  MoveAbsJ [[135.73,-26.28,-187.24,-106.91,-52.79,56.60],[9E9,9E9,9E9,9E9,9E9,9E9]],speeddata0,DefaultBlend,tool0;
  MoveAbsJ [[136.14,-26.36,-187.04,-105.92,-52.94,56.91],[9E9,9E9,9E9,9E9,9E9,9E9]],speeddata0,DefaultBlend,tool0;
  MoveAbsJ [[136.55,-26.45,-186.84,-104.93,-53.08,57.22],[9E9,9E9,9E9,9E9,9E9,9E9]],speeddata0,DefaultBlend,tool0;
  MoveAbsJ [[136.96,-26.54,-186.65,-103.94,-53.23,57.53],[9E9,9E9,9E9,9E9,9E9,9E9]],speeddata0,DefaultBlend,tool0;
  MoveAbsJ [[137.37,-26.63,-186.45,-102.95,-53.37,57.84],[9E9,9E9,9E9,9E9,9E9,9E9]],speeddata0,DefaultBlend,tool0;
  MoveAbsJ [[137.78,-26.71,-186.25,-101.96,-53.52,58.14],[9E9,9E9,9E9,9E9,9E9,9E9]],speeddata0,DefaultBlend,tool0;
  MoveAbsJ [[138.19,-26.80,-186.05,-100.97,-53.66,58.45],[9E9,9E9,9E9,9E9,9E9,9E9]],speeddata0,DefaultBlend,tool0;
  MoveAbsJ [[138.60,-26.89,-185.85,-99.98,-53.81,58.76],[9E9,9E9,9E9,9E9,9E9,9E9]],speeddata0,DefaultBlend,tool0;
  MoveAbsJ [[139.01,-26.97,-185.66,-98.99,-53.95,59.07],[9E9,9E9,9E9,9E9,9E9,9E9]],speeddata0,DefaultBlend,tool0;
  MoveAbsJ [[139.42,-27.06,-185.46,-98.00,-54.10,59.38],[9E9,9E9,9E9,9E9,9E9,9E9]],speeddata0,DefaultBlend,tool0;
  MoveAbsJ [[139.83,-27.15,-185.26,-97.01,-54.24,59.69],[9E9,9E9,9E9,9E9,9E9,9E9]],speeddata0,DefaultBlend,tool0;
  MoveAbsJ [[140.24,-27.23,-185.06,-96.02,-54.39,60.00],[9E9,9E9,9E9,9E9,9E9,9E9]],speeddata0,DefaultBlend,tool0;
  MoveAbsJ [[140.65,-27.32,-184.86,-95.03,-54.53,60.31],[9E9,9E9,9E9,9E9,9E9,9E9]],speeddata0,DefaultBlend,tool0;
  MoveAbsJ [[141.06,-27.41,-184.67,-94.04,-54.68,60.62],[9E9,9E9,9E9,9E9,9E9,9E9]],speeddata0,DefaultBlend,tool0;
  MoveAbsJ [[141.47,-27.49,-184.47,-93.05,-54.83,60.93],[9E9,9E9,9E9,9E9,9E9,9E9]],speeddata0,DefaultBlend,tool0;
  MoveAbsJ [[141.88,-27.58,-184.27,-92.06,-54.97,61.24],[9E9,9E9,9E9,9E9,9E9,9E9]],speeddata0,DefaultBlend,tool0;
  MoveAbsJ [[142.29,-27.67,-184.07,-91.07,-55.12,61.55],[9E9,9E9,9E9,9E9,9E9,9E9]],speeddata0,DefaultBlend,tool0;
  MoveAbsJ [[142.70,-27.75,-183.87,-90.08,-55.26,61.86],[9E9,9E9,9E9,9E9,9E9,9E9]],speeddata0,DefaultBlend,tool0;
  MoveAbsJ [[143.11,-27.84,-183.68,-89.09,-55.41,62.17],[9E9,9E9,9E9,9E9,9E9,9E9]],speeddata0,DefaultBlend,tool0;
  MoveAbsJ [[143.52,-27.93,-183.48,-88.10,-55.55,62.47],[9E9,9E9,9E9,9E9,9E9,9E9]],speeddata0,DefaultBlend,tool0;
  MoveAbsJ [[143.93,-28.01,-183.28,-87.11,-55.70,62.78],[9E9,9E9,9E9,9E9,9E9,9E9]],speeddata0,DefaultBlend,tool0;
  MoveAbsJ [[144.34,-28.10,-183.08,-86.12,-55.84,63.09],[9E9,9E9,9E9,9E9,9E9,9E9]],speeddata0,DefaultBlend,tool0;
  MoveAbsJ [[144.75,-28.19,-182.88,-85.13,-55.99,63.40],[9E9,9E9,9E9,9E9,9E9,9E9]],speeddata0,DefaultBlend,tool0;
  MoveAbsJ [[145.16,-28.27,-182.69,-84.14,-56.13,63.71],[9E9,9E9,9E9,9E9,9E9,9E9]],speeddata0,DefaultBlend,tool0;
  MoveAbsJ [[145.57,-28.36,-182.49,-83.15,-56.28,64.02],[9E9,9E9,9E9,9E9,9E9,9E9]],speeddata0,DefaultBlend,tool0;
  MoveAbsJ [[145.98,-28.45,-182.29,-82.16,-56.42,64.33],[9E9,9E9,9E9,9E9,9E9,9E9]],speeddata0,DefaultBlend,tool0;
  MoveAbsJ [[146.39,-28.54,-182.09,-81.17,-56.57,64.64],[9E9,9E9,9E9,9E9,9E9,9E9]],speeddata0,DefaultBlend,tool0;
  MoveAbsJ [[146.80,-28.62,-181.90,-80.18,-56.72,64.95],[9E9,9E9,9E9,9E9,9E9,9E9]],speeddata0,DefaultBlend,tool0;
  MoveAbsJ [[147.21,-28.71,-181.70,-79.19,-56.86,65.26],[9E9,9E9,9E9,9E9,9E9,9E9]],speeddata0,DefaultBlend,tool0;
  MoveAbsJ [[147.62,-28.80,-181.50,-78.20,-57.01,65.57],[9E9,9E9,9E9,9E9,9E9,9E9]],speeddata0,DefaultBlend,tool0;
  MoveAbsJ [[148.03,-28.88,-181.30,-77.21,-57.15,65.88],[9E9,9E9,9E9,9E9,9E9,9E9]],speeddata0,DefaultBlend,tool0;
  MoveAbsJ [[148.44,-28.97,-181.10,-76.23,-57.30,66.19],[9E9,9E9,9E9,9E9,9E9,9E9]],speeddata0,DefaultBlend,tool0;
  MoveAbsJ [[148.85,-29.06,-180.91,-75.24,-57.44,66.49],[9E9,9E9,9E9,9E9,9E9,9E9]],speeddata0,DefaultBlend,tool0;
  MoveAbsJ [[149.26,-29.14,-180.71,-74.25,-57.59,66.80],[9E9,9E9,9E9,9E9,9E9,9E9]],speeddata0,DefaultBlend,tool0;
  MoveAbsJ [[149.67,-29.23,-180.51,-73.26,-57.73,67.11],[9E9,9E9,9E9,9E9,9E9,9E9]],speeddata0,DefaultBlend,tool0;
  MoveAbsJ [[150.08,-29.32,-180.31,-72.27,-57.88,67.42],[9E9,9E9,9E9,9E9,9E9,9E9]],speeddata0,DefaultBlend,tool0;
  MoveAbsJ [[150.49,-29.40,-180.11,-71.28,-58.02,67.73],[9E9,9E9,9E9,9E9,9E9,9E9]],speeddata0,DefaultBlend,tool0;
  MoveAbsJ [[150.90,-29.49,-179.92,-70.29,-58.17,68.04],[9E9,9E9,9E9,9E9,9E9,9E9]],speeddata0,DefaultBlend,tool0;
  MoveAbsJ [[151.31,-29.58,-179.72,-69.30,-58.31,68.35],[9E9,9E9,9E9,9E9,9E9,9E9]],speeddata0,DefaultBlend,tool0;
  MoveAbsJ [[151.72,-29.66,-179.52,-68.31,-58.46,68.66],[9E9,9E9,9E9,9E9,9E9,9E9]],speeddata0,DefaultBlend,tool0;
  MoveAbsJ [[152.13,-29.75,-179.32,-67.32,-58.61,68.97],[9E9,9E9,9E9,9E9,9E9,9E9]],speeddata0,DefaultBlend,tool0;
  MoveAbsJ [[152.54,-29.84,-179.12,-66.33,-58.75,69.28],[9E9,9E9,9E9,9E9,9E9,9E9]],speeddata0,DefaultBlend,tool0;
  MoveAbsJ [[152.95,-29.92,-178.93,-65.34,-58.90,69.59],[9E9,9E9,9E9,9E9,9E9,9E9]],speeddata0,DefaultBlend,tool0;
  MoveAbsJ [[153.36,-30.01,-178.73,-64.35,-59.04,69.90],[9E9,9E9,9E9,9E9,9E9,9E9]],speeddata0,DefaultBlend,tool0;
  MoveAbsJ [[153.77,-30.10,-178.53,-63.36,-59.19,70.21],[9E9,9E9,9E9,9E9,9E9,9E9]],speeddata0,DefaultBlend,tool0;
  MoveAbsJ [[154.18,-30.18,-178.33,-62.37,-59.33,70.51],[9E9,9E9,9E9,9E9,9E9,9E9]],speeddata0,DefaultBlend,tool0;
  MoveAbsJ [[154.59,-30.27,-178.13,-61.38,-59.48,70.82],[9E9,9E9,9E9,9E9,9E9,9E9]],speeddata0,DefaultBlend,tool0;
  MoveAbsJ [[155.00,-30.36,-177.94,-60.39,-59.62,71.13],[9E9,9E9,9E9,9E9,9E9,9E9]],speeddata0,DefaultBlend,tool0;
  MoveAbsJ [[155.40,-30.44,-177.74,-59.40,-59.77,71.44],[9E9,9E9,9E9,9E9,9E9,9E9]],speeddata0,DefaultBlend,tool0;
  MoveAbsJ [[155.81,-30.53,-177.54,-58.41,-59.91,71.75],[9E9,9E9,9E9,9E9,9E9,9E9]],speeddata0,DefaultBlend,tool0;
  MoveAbsJ [[156.22,-30.62,-177.34,-57.42,-60.06,72.06],[9E9,9E9,9E9,9E9,9E9,9E9]],speeddata0,DefaultBlend,tool0;
  MoveAbsJ [[156.63,-30.71,-177.14,-56.43,-60.21,72.37],[9E9,9E9,9E9,9E9,9E9,9E9]],speeddata0,DefaultBlend,tool0;
  MoveAbsJ [[157.04,-30.79,-176.95,-55.44,-60.35,72.68],[9E9,9E9,9E9,9E9,9E9,9E9]],speeddata0,DefaultBlend,tool0;
  MoveAbsJ [[157.45,-30.88,-176.75,-54.45,-60.50,72.99],[9E9,9E9,9E9,9E9,9E9,9E9]],speeddata0,DefaultBlend,tool0;
  MoveAbsJ [[157.86,-30.97,-176.55,-53.46,-60.64,73.30],[9E9,9E9,9E9,9E9,9E9,9E9]],speeddata0,DefaultBlend,tool0;
  MoveAbsJ [[158.27,-31.05,-176.35,-52.47,-60.79,73.61],[9E9,9E9,9E9,9E9,9E9,9E9]],speeddata0,DefaultBlend,tool0;
  MoveAbsJ [[158.68,-31.14,-176.16,-51.48,-60.93,73.92],[9E9,9E9,9E9,9E9,9E9,9E9]],speeddata0,DefaultBlend,tool0;
  MoveAbsJ [[159.09,-31.23,-175.96,-50.49,-61.08,74.23],[9E9,9E9,9E9,9E9,9E9,9E9]],speeddata0,DefaultBlend,tool0;
  MoveAbsJ [[159.50,-31.31,-175.76,-49.50,-61.22,74.53],[9E9,9E9,9E9,9E9,9E9,9E9]],speeddata0,DefaultBlend,tool0;
  MoveAbsJ [[159.91,-31.40,-175.56,-48.51,-61.37,74.84],[9E9,9E9,9E9,9E9,9E9,9E9]],speeddata0,DefaultBlend,tool0;
  MoveAbsJ [[160.32,-31.49,-175.36,-47.52,-61.51,75.15],[9E9,9E9,9E9,9E9,9E9,9E9]],speeddata0,DefaultBlend,tool0;
  MoveAbsJ [[160.73,-31.57,-175.17,-46.53,-61.66,75.46],[9E9,9E9,9E9,9E9,9E9,9E9]],speeddata0,DefaultBlend,tool0;
  MoveAbsJ [[161.14,-31.66,-174.97,-45.54,-61.80,75.77],[9E9,9E9,9E9,9E9,9E9,9E9]],speeddata0,DefaultBlend,tool0;
  MoveAbsJ [[161.55,-31.75,-174.77,-44.55,-61.95,76.08],[9E9,9E9,9E9,9E9,9E9,9E9]],speeddata0,DefaultBlend,tool0;
  MoveAbsJ [[161.96,-31.83,-174.57,-43.56,-62.10,76.39],[9E9,9E9,9E9,9E9,9E9,9E9]],speeddata0,DefaultBlend,tool0;
  MoveAbsJ [[162.37,-31.92,-174.37,-42.57,-62.24,76.70],[9E9,9E9,9E9,9E9,9E9,9E9]],speeddata0,DefaultBlend,tool0;
  MoveAbsJ [[162.78,-32.01,-174.18,-41.58,-62.39,77.01],[9E9,9E9,9E9,9E9,9E9,9E9]],speeddata0,DefaultBlend,tool0;
  MoveAbsJ [[163.19,-32.09,-173.98,-40.59,-62.53,77.32],[9E9,9E9,9E9,9E9,9E9,9E9]],speeddata0,DefaultBlend,tool0;
  MoveAbsJ [[163.60,-32.18,-173.78,-39.60,-62.68,77.63],[9E9,9E9,9E9,9E9,9E9,9E9]],speeddata0,DefaultBlend,tool0;
  MoveAbsJ [[164.01,-32.27,-173.58,-38.61,-62.82,77.94],[9E9,9E9,9E9,9E9,9E9,9E9]],speeddata0,DefaultBlend,tool0;
  MoveAbsJ [[164.42,-32.35,-173.38,-37.62,-62.97,78.25],[9E9,9E9,9E9,9E9,9E9,9E9]],speeddata0,DefaultBlend,tool0;
  MoveAbsJ [[164.83,-32.44,-173.19,-36.63,-63.11,78.56],[9E9,9E9,9E9,9E9,9E9,9E9]],speeddata0,DefaultBlend,tool0;
  MoveAbsJ [[165.24,-32.53,-172.99,-35.64,-63.26,78.86],[9E9,9E9,9E9,9E9,9E9,9E9]],speeddata0,DefaultBlend,tool0;
  MoveAbsJ [[165.65,-32.61,-172.79,-34.65,-63.40,79.17],[9E9,9E9,9E9,9E9,9E9,9E9]],speeddata0,DefaultBlend,tool0;
  MoveAbsJ [[166.06,-32.70,-172.59,-33.66,-63.55,79.48],[9E9,9E9,9E9,9E9,9E9,9E9]],speeddata0,DefaultBlend,tool0;
  MoveAbsJ [[166.47,-32.79,-172.39,-32.67,-63.69,79.79],[9E9,9E9,9E9,9E9,9E9,9E9]],speeddata0,DefaultBlend,tool0;
  MoveAbsJ [[166.88,-32.88,-172.20,-31.68,-63.84,80.10],[9E9,9E9,9E9,9E9,9E9,9E9]],speeddata0,DefaultBlend,tool0;
  MoveAbsJ [[167.29,-32.96,-172.00,-30.69,-63.99,80.41],[9E9,9E9,9E9,9E9,9E9,9E9]],speeddata0,DefaultBlend,tool0;
  MoveAbsJ [[167.70,-33.05,-171.80,-29.70,-64.13,80.72],[9E9,9E9,9E9,9E9,9E9,9E9]],speeddata0,DefaultBlend,tool0;
  MoveAbsJ [[168.11,-33.14,-171.60,-28.71,-64.28,81.03],[9E9,9E9,9E9,9E9,9E9,9E9]],speeddata0,DefaultBlend,tool0;
  MoveAbsJ [[168.52,-33.22,-171.40,-27.72,-64.42,81.34],[9E9,9E9,9E9,9E9,9E9,9E9]],speeddata0,DefaultBlend,tool0;
  MoveAbsJ [[168.93,-33.31,-171.21,-26.73,-64.57,81.65],[9E9,9E9,9E9,9E9,9E9,9E9]],speeddata0,DefaultBlend,tool0;
  MoveAbsJ [[169.34,-33.40,-171.01,-25.74,-64.71,81.96],[9E9,9E9,9E9,9E9,9E9,9E9]],speeddata0,DefaultBlend,tool0;
  MoveAbsJ [[169.75,-33.48,-170.81,-24.75,-64.86,82.27],[9E9,9E9,9E9,9E9,9E9,9E9]],speeddata0,DefaultBlend,tool0;
  MoveAbsJ [[170.16,-33.57,-170.61,-23.76,-65.00,82.58],[9E9,9E9,9E9,9E9,9E9,9E9]],speeddata0,DefaultBlend,tool0;
  MoveAbsJ [[170.57,-33.66,-170.42,-22.77,-65.15,82.88],[9E9,9E9,9E9,9E9,9E9,9E9]],speeddata0,DefaultBlend,tool0;
  MoveAbsJ [[170.98,-33.74,-170.22,-21.78,-65.29,83.19],[9E9,9E9,9E9,9E9,9E9,9E9]],speeddata0,DefaultBlend,tool0;
  MoveAbsJ [[171.39,-33.83,-170.02,-20.79,-65.44,83.50],[9E9,9E9,9E9,9E9,9E9,9E9]],speeddata0,DefaultBlend,tool0;
  MoveAbsJ [[171.80,-33.92,-169.82,-19.80,-65.58,83.81],[9E9,9E9,9E9,9E9,9E9,9E9]],speeddata0,DefaultBlend,tool0;
  MoveAbsJ [[172.21,-34.00,-169.62,-18.81,-65.73,84.12],[9E9,9E9,9E9,9E9,9E9,9E9]],speeddata0,DefaultBlend,tool0;
  MoveAbsJ [[172.62,-34.09,-169.43,-17.82,-65.88,84.43],[9E9,9E9,9E9,9E9,9E9,9E9]],speeddata0,DefaultBlend,tool0;
  MoveAbsJ [[173.03,-34.18,-169.23,-16.83,-66.02,84.74],[9E9,9E9,9E9,9E9,9E9,9E9]],speeddata0,DefaultBlend,tool0;
  MoveAbsJ [[173.44,-34.26,-169.03,-15.84,-66.17,85.05],[9E9,9E9,9E9,9E9,9E9,9E9]],speeddata0,DefaultBlend,tool0;
  MoveAbsJ [[173.85,-34.35,-168.83,-14.85,-66.31,85.36],[9E9,9E9,9E9,9E9,9E9,9E9]],speeddata0,DefaultBlend,tool0;
  MoveAbsJ [[174.26,-34.44,-168.63,-13.86,-66.46,85.67],[9E9,9E9,9E9,9E9,9E9,9E9]],speeddata0,DefaultBlend,tool0;
  MoveAbsJ [[174.67,-34.52,-168.44,-12.87,-66.60,85.98],[9E9,9E9,9E9,9E9,9E9,9E9]],speeddata0,DefaultBlend,tool0;
  MoveAbsJ [[175.08,-34.61,-168.24,-11.88,-66.75,86.29],[9E9,9E9,9E9,9E9,9E9,9E9]],speeddata0,DefaultBlend,tool0;
  MoveAbsJ [[175.49,-34.70,-168.04,-10.89,-66.89,86.60],[9E9,9E9,9E9,9E9,9E9,9E9]],speeddata0,DefaultBlend,tool0;
  MoveAbsJ [[175.90,-34.78,-167.84,-9.90,-67.04,86.90],[9E9,9E9,9E9,9E9,9E9,9E9]],speeddata0,DefaultBlend,tool0;
  MoveAbsJ [[176.31,-34.87,-167.64,-8.91,-67.18,87.21],[9E9,9E9,9E9,9E9,9E9,9E9]],speeddata0,DefaultBlend,tool0;
  MoveAbsJ [[176.72,-34.96,-167.45,-7.92,-67.33,87.52],[9E9,9E9,9E9,9E9,9E9,9E9]],speeddata0,DefaultBlend,tool0;
  MoveAbsJ [[177.13,-35.05,-167.25,-6.93,-67.47,87.83],[9E9,9E9,9E9,9E9,9E9,9E9]],speeddata0,DefaultBlend,tool0;
  MoveAbsJ [[177.54,-35.13,-167.05,-5.94,-67.62,88.14],[9E9,9E9,9E9,9E9,9E9,9E9]],speeddata0,DefaultBlend,tool0;
  MoveAbsJ [[177.95,-35.22,-166.85,-4.95,-67.77,88.45],[9E9,9E9,9E9,9E9,9E9,9E9]],speeddata0,DefaultBlend,tool0;
  MoveAbsJ [[178.36,-35.31,-166.65,-3.96,-67.91,88.76],[9E9,9E9,9E9,9E9,9E9,9E9]],speeddata0,DefaultBlend,tool0;
  MoveAbsJ [[178.77,-35.39,-166.46,-2.97,-68.06,89.07],[9E9,9E9,9E9,9E9,9E9,9E9]],speeddata0,DefaultBlend,tool0;
  MoveAbsJ [[179.18,-35.48,-166.26,-1.98,-68.20,89.38],[9E9,9E9,9E9,9E9,9E9,9E9]],speeddata0,DefaultBlend,tool0;
  MoveAbsJ [[179.59,-35.57,-166.06,-0.99,-68.35,89.69],[9E9,9E9,9E9,9E9,9E9,9E9]],speeddata0,DefaultBlend,tool0;
  MoveAbsJ [[180.00,-35.65,-165.86,0.00,-68.49,90.00],[9E9,9E9,9E9,9E9,9E9,9E9]],speeddata0,FinePoint,tool0;
  TPWrite "Action 18 LinearMovement.";
  MoveAbsJ [[180.00,-35.65,-165.86,0.00,-68.49,90.00],[9E9,9E9,9E9,9E9,9E9,9E9]],speeddata0,DefaultBlend,tool0;
  MoveAbsJ [[180.00,-35.59,-165.97,0.00,-68.44,90.00],[9E9,9E9,9E9,9E9,9E9,9E9]],speeddata0,DefaultBlend,tool0;
  MoveAbsJ [[180.00,-36.29,-166.18,0.00,-67.54,90.00],[9E9,9E9,9E9,9E9,9E9,9E9]],speeddata0,DefaultBlend,tool0;
  MoveAbsJ [[180.00,-37.00,-166.36,0.00,-66.64,90.00],[9E9,9E9,9E9,9E9,9E9,9E9]],speeddata0,DefaultBlend,tool0;
  MoveAbsJ [[180.00,-37.73,-166.51,0.00,-65.76,90.00],[9E9,9E9,9E9,9E9,9E9,9E9]],speeddata0,DefaultBlend,tool0;
  MoveAbsJ [[180.00,-38.47,-166.65,0.00,-64.88,90.00],[9E9,9E9,9E9,9E9,9E9,9E9]],speeddata0,DefaultBlend,tool0;
  MoveAbsJ [[180.00,-39.22,-166.76,0.00,-64.02,90.00],[9E9,9E9,9E9,9E9,9E9,9E9]],speeddata0,DefaultBlend,tool0;
  MoveAbsJ [[180.00,-39.99,-166.85,0.00,-63.16,90.00],[9E9,9E9,9E9,9E9,9E9,9E9]],speeddata0,DefaultBlend,tool0;
  MoveAbsJ [[180.00,-40.78,-166.91,0.00,-62.31,90.00],[9E9,9E9,9E9,9E9,9E9,9E9]],speeddata0,DefaultBlend,tool0;
  MoveAbsJ [[180.00,-41.57,-166.96,0.00,-61.47,90.00],[9E9,9E9,9E9,9E9,9E9,9E9]],speeddata0,FinePoint,tool0;
  TPWrite "Action 19 OpenGripper.";
  TPWrite "Press Play to Continue";
  Stop;
  TPWrite "Action 20 LinearMovement.";
  MoveAbsJ [[180.00,-41.57,-166.96,-0.00,-61.47,90.00],[9E9,9E9,9E9,9E9,9E9,9E9]],speeddata0,DefaultBlend,tool0;
  MoveAbsJ [[180.00,-40.78,-166.92,0.00,-62.30,90.00],[9E9,9E9,9E9,9E9,9E9,9E9]],speeddata0,DefaultBlend,tool0;
  MoveAbsJ [[180.00,-39.99,-166.86,0.00,-63.14,90.00],[9E9,9E9,9E9,9E9,9E9,9E9]],speeddata0,DefaultBlend,tool0;
  MoveAbsJ [[180.00,-39.22,-166.78,0.00,-64.00,90.00],[9E9,9E9,9E9,9E9,9E9,9E9]],speeddata0,DefaultBlend,tool0;
  MoveAbsJ [[180.00,-38.46,-166.67,0.00,-64.86,90.00],[9E9,9E9,9E9,9E9,9E9,9E9]],speeddata0,DefaultBlend,tool0;
  MoveAbsJ [[180.00,-37.72,-166.54,0.00,-65.74,90.00],[9E9,9E9,9E9,9E9,9E9,9E9]],speeddata0,DefaultBlend,tool0;
  MoveAbsJ [[180.00,-36.99,-166.39,0.00,-66.63,90.00],[9E9,9E9,9E9,9E9,9E9,9E9]],speeddata0,DefaultBlend,tool0;
  MoveAbsJ [[180.00,-36.27,-166.21,0.00,-67.52,90.00],[9E9,9E9,9E9,9E9,9E9,9E9]],speeddata0,DefaultBlend,tool0;
  MoveAbsJ [[180.00,-35.58,-166.00,0.00,-68.42,90.00],[9E9,9E9,9E9,9E9,9E9,9E9]],speeddata0,FinePoint,tool0;
  TPWrite "Action 21 FreeMovement.";
  MoveAbsJ [[180.00,-35.58,-166.00,0.00,-68.42,90.00],[9E9,9E9,9E9,9E9,9E9,9E9]],speeddata0,DefaultBlend,tool0;
  MoveAbsJ [[179.59,-35.49,-166.20,-0.99,-68.28,89.69],[9E9,9E9,9E9,9E9,9E9,9E9]],speeddata0,DefaultBlend,tool0;
  MoveAbsJ [[179.18,-35.40,-166.40,-1.98,-68.13,89.38],[9E9,9E9,9E9,9E9,9E9,9E9]],speeddata0,DefaultBlend,tool0;
  MoveAbsJ [[178.77,-35.32,-166.59,-2.97,-67.99,89.07],[9E9,9E9,9E9,9E9,9E9,9E9]],speeddata0,DefaultBlend,tool0;
  MoveAbsJ [[178.36,-35.23,-166.79,-3.96,-67.84,88.76],[9E9,9E9,9E9,9E9,9E9,9E9]],speeddata0,DefaultBlend,tool0;
  MoveAbsJ [[177.95,-35.14,-166.99,-4.95,-67.70,88.45],[9E9,9E9,9E9,9E9,9E9,9E9]],speeddata0,DefaultBlend,tool0;
  MoveAbsJ [[177.54,-35.06,-167.18,-5.94,-67.55,88.14],[9E9,9E9,9E9,9E9,9E9,9E9]],speeddata0,DefaultBlend,tool0;
  MoveAbsJ [[177.13,-34.97,-167.38,-6.93,-67.41,87.83],[9E9,9E9,9E9,9E9,9E9,9E9]],speeddata0,DefaultBlend,tool0;
  MoveAbsJ [[176.72,-34.89,-167.58,-7.92,-67.26,87.52],[9E9,9E9,9E9,9E9,9E9,9E9]],speeddata0,DefaultBlend,tool0;
  MoveAbsJ [[176.31,-34.80,-167.77,-8.91,-67.12,87.21],[9E9,9E9,9E9,9E9,9E9,9E9]],speeddata0,DefaultBlend,tool0;
  MoveAbsJ [[175.90,-34.71,-167.97,-9.90,-66.97,86.91],[9E9,9E9,9E9,9E9,9E9,9E9]],speeddata0,DefaultBlend,tool0;
  MoveAbsJ [[175.49,-34.63,-168.17,-10.89,-66.83,86.60],[9E9,9E9,9E9,9E9,9E9,9E9]],speeddata0,DefaultBlend,tool0;
  MoveAbsJ [[175.08,-34.54,-168.36,-11.88,-66.68,86.29],[9E9,9E9,9E9,9E9,9E9,9E9]],speeddata0,DefaultBlend,tool0;
  MoveAbsJ [[174.67,-34.45,-168.56,-12.87,-66.54,85.98],[9E9,9E9,9E9,9E9,9E9,9E9]],speeddata0,DefaultBlend,tool0;
  MoveAbsJ [[174.26,-34.37,-168.76,-13.86,-66.39,85.67],[9E9,9E9,9E9,9E9,9E9,9E9]],speeddata0,DefaultBlend,tool0;
  MoveAbsJ [[173.85,-34.28,-168.95,-14.85,-66.25,85.36],[9E9,9E9,9E9,9E9,9E9,9E9]],speeddata0,DefaultBlend,tool0;
  MoveAbsJ [[173.44,-34.20,-169.15,-15.84,-66.10,85.05],[9E9,9E9,9E9,9E9,9E9,9E9]],speeddata0,DefaultBlend,tool0;
  MoveAbsJ [[173.03,-34.11,-169.35,-16.83,-65.96,84.74],[9E9,9E9,9E9,9E9,9E9,9E9]],speeddata0,DefaultBlend,tool0;
  MoveAbsJ [[172.62,-34.02,-169.54,-17.82,-65.81,84.43],[9E9,9E9,9E9,9E9,9E9,9E9]],speeddata0,DefaultBlend,tool0;
  MoveAbsJ [[172.21,-33.94,-169.74,-18.81,-65.67,84.12],[9E9,9E9,9E9,9E9,9E9,9E9]],speeddata0,DefaultBlend,tool0;
  MoveAbsJ [[171.80,-33.85,-169.94,-19.80,-65.52,83.81],[9E9,9E9,9E9,9E9,9E9,9E9]],speeddata0,DefaultBlend,tool0;
  MoveAbsJ [[171.39,-33.76,-170.13,-20.78,-65.38,83.50],[9E9,9E9,9E9,9E9,9E9,9E9]],speeddata0,DefaultBlend,tool0;
  MoveAbsJ [[170.98,-33.68,-170.33,-21.77,-65.23,83.19],[9E9,9E9,9E9,9E9,9E9,9E9]],speeddata0,DefaultBlend,tool0;
  MoveAbsJ [[170.57,-33.59,-170.53,-22.76,-65.09,82.88],[9E9,9E9,9E9,9E9,9E9,9E9]],speeddata0,DefaultBlend,tool0;
  MoveAbsJ [[170.16,-33.51,-170.73,-23.75,-64.94,82.57],[9E9,9E9,9E9,9E9,9E9,9E9]],speeddata0,DefaultBlend,tool0;
  MoveAbsJ [[169.75,-33.42,-170.92,-24.74,-64.80,82.26],[9E9,9E9,9E9,9E9,9E9,9E9]],speeddata0,DefaultBlend,tool0;
  MoveAbsJ [[169.34,-33.33,-171.12,-25.73,-64.65,81.95],[9E9,9E9,9E9,9E9,9E9,9E9]],speeddata0,DefaultBlend,tool0;
  MoveAbsJ [[168.93,-33.25,-171.32,-26.72,-64.51,81.64],[9E9,9E9,9E9,9E9,9E9,9E9]],speeddata0,DefaultBlend,tool0;
  MoveAbsJ [[168.53,-33.16,-171.51,-27.71,-64.36,81.34],[9E9,9E9,9E9,9E9,9E9,9E9]],speeddata0,DefaultBlend,tool0;
  MoveAbsJ [[168.12,-33.07,-171.71,-28.70,-64.22,81.03],[9E9,9E9,9E9,9E9,9E9,9E9]],speeddata0,DefaultBlend,tool0;
  MoveAbsJ [[167.71,-32.99,-171.91,-29.69,-64.08,80.72],[9E9,9E9,9E9,9E9,9E9,9E9]],speeddata0,DefaultBlend,tool0;
  MoveAbsJ [[167.30,-32.90,-172.10,-30.68,-63.93,80.41],[9E9,9E9,9E9,9E9,9E9,9E9]],speeddata0,DefaultBlend,tool0;
  MoveAbsJ [[166.89,-32.82,-172.30,-31.67,-63.79,80.10],[9E9,9E9,9E9,9E9,9E9,9E9]],speeddata0,DefaultBlend,tool0;
  MoveAbsJ [[166.48,-32.73,-172.50,-32.66,-63.64,79.79],[9E9,9E9,9E9,9E9,9E9,9E9]],speeddata0,DefaultBlend,tool0;
  MoveAbsJ [[166.07,-32.64,-172.69,-33.65,-63.50,79.48],[9E9,9E9,9E9,9E9,9E9,9E9]],speeddata0,DefaultBlend,tool0;
  MoveAbsJ [[165.66,-32.56,-172.89,-34.64,-63.35,79.17],[9E9,9E9,9E9,9E9,9E9,9E9]],speeddata0,DefaultBlend,tool0;
  MoveAbsJ [[165.25,-32.47,-173.09,-35.63,-63.21,78.86],[9E9,9E9,9E9,9E9,9E9,9E9]],speeddata0,DefaultBlend,tool0;
  MoveAbsJ [[164.84,-32.38,-173.28,-36.62,-63.06,78.55],[9E9,9E9,9E9,9E9,9E9,9E9]],speeddata0,DefaultBlend,tool0;
  MoveAbsJ [[164.43,-32.30,-173.48,-37.61,-62.92,78.24],[9E9,9E9,9E9,9E9,9E9,9E9]],speeddata0,DefaultBlend,tool0;
  MoveAbsJ [[164.02,-32.21,-173.68,-38.60,-62.77,77.93],[9E9,9E9,9E9,9E9,9E9,9E9]],speeddata0,DefaultBlend,tool0;
  MoveAbsJ [[163.61,-32.13,-173.87,-39.59,-62.63,77.62],[9E9,9E9,9E9,9E9,9E9,9E9]],speeddata0,DefaultBlend,tool0;
  MoveAbsJ [[163.20,-32.04,-174.07,-40.58,-62.48,77.31],[9E9,9E9,9E9,9E9,9E9,9E9]],speeddata0,DefaultBlend,tool0;
  MoveAbsJ [[162.79,-31.95,-174.27,-41.57,-62.34,77.00],[9E9,9E9,9E9,9E9,9E9,9E9]],speeddata0,DefaultBlend,tool0;
  MoveAbsJ [[162.38,-31.87,-174.46,-42.56,-62.19,76.69],[9E9,9E9,9E9,9E9,9E9,9E9]],speeddata0,DefaultBlend,tool0;
  MoveAbsJ [[161.97,-31.78,-174.66,-43.55,-62.05,76.38],[9E9,9E9,9E9,9E9,9E9,9E9]],speeddata0,DefaultBlend,tool0;
  MoveAbsJ [[161.56,-31.69,-174.86,-44.54,-61.90,76.07],[9E9,9E9,9E9,9E9,9E9,9E9]],speeddata0,DefaultBlend,tool0;
  MoveAbsJ [[161.15,-31.61,-175.05,-45.53,-61.76,75.76],[9E9,9E9,9E9,9E9,9E9,9E9]],speeddata0,DefaultBlend,tool0;
  MoveAbsJ [[160.74,-31.52,-175.25,-46.52,-61.61,75.46],[9E9,9E9,9E9,9E9,9E9,9E9]],speeddata0,DefaultBlend,tool0;
  MoveAbsJ [[160.33,-31.44,-175.45,-47.51,-61.47,75.15],[9E9,9E9,9E9,9E9,9E9,9E9]],speeddata0,DefaultBlend,tool0;
  MoveAbsJ [[159.92,-31.35,-175.64,-48.50,-61.32,74.84],[9E9,9E9,9E9,9E9,9E9,9E9]],speeddata0,DefaultBlend,tool0;
  MoveAbsJ [[159.51,-31.26,-175.84,-49.49,-61.18,74.53],[9E9,9E9,9E9,9E9,9E9,9E9]],speeddata0,DefaultBlend,tool0;
  MoveAbsJ [[159.10,-31.18,-176.04,-50.48,-61.03,74.22],[9E9,9E9,9E9,9E9,9E9,9E9]],speeddata0,DefaultBlend,tool0;
  MoveAbsJ [[158.69,-31.09,-176.24,-51.47,-60.89,73.91],[9E9,9E9,9E9,9E9,9E9,9E9]],speeddata0,DefaultBlend,tool0;
  MoveAbsJ [[158.28,-31.00,-176.43,-52.46,-60.74,73.60],[9E9,9E9,9E9,9E9,9E9,9E9]],speeddata0,DefaultBlend,tool0;
  MoveAbsJ [[157.87,-30.92,-176.63,-53.45,-60.60,73.29],[9E9,9E9,9E9,9E9,9E9,9E9]],speeddata0,DefaultBlend,tool0;
  MoveAbsJ [[157.46,-30.83,-176.83,-54.44,-60.45,72.98],[9E9,9E9,9E9,9E9,9E9,9E9]],speeddata0,DefaultBlend,tool0;
  MoveAbsJ [[157.05,-30.75,-177.02,-55.43,-60.31,72.67],[9E9,9E9,9E9,9E9,9E9,9E9]],speeddata0,DefaultBlend,tool0;
  MoveAbsJ [[156.64,-30.66,-177.22,-56.42,-60.16,72.36],[9E9,9E9,9E9,9E9,9E9,9E9]],speeddata0,DefaultBlend,tool0;
  MoveAbsJ [[156.23,-30.57,-177.42,-57.41,-60.02,72.05],[9E9,9E9,9E9,9E9,9E9,9E9]],speeddata0,DefaultBlend,tool0;
  MoveAbsJ [[155.82,-30.49,-177.61,-58.40,-59.87,71.74],[9E9,9E9,9E9,9E9,9E9,9E9]],speeddata0,DefaultBlend,tool0;
  MoveAbsJ [[155.41,-30.40,-177.81,-59.39,-59.73,71.43],[9E9,9E9,9E9,9E9,9E9,9E9]],speeddata0,DefaultBlend,tool0;
  MoveAbsJ [[155.00,-30.31,-178.01,-60.38,-59.58,71.12],[9E9,9E9,9E9,9E9,9E9,9E9]],speeddata0,DefaultBlend,tool0;
  MoveAbsJ [[154.59,-30.23,-178.20,-61.36,-59.44,70.81],[9E9,9E9,9E9,9E9,9E9,9E9]],speeddata0,DefaultBlend,tool0;
  MoveAbsJ [[154.18,-30.14,-178.40,-62.35,-59.29,70.50],[9E9,9E9,9E9,9E9,9E9,9E9]],speeddata0,DefaultBlend,tool0;
  MoveAbsJ [[153.77,-30.06,-178.60,-63.34,-59.15,70.19],[9E9,9E9,9E9,9E9,9E9,9E9]],speeddata0,DefaultBlend,tool0;
  MoveAbsJ [[153.36,-29.97,-178.79,-64.33,-59.01,69.89],[9E9,9E9,9E9,9E9,9E9,9E9]],speeddata0,DefaultBlend,tool0;
  MoveAbsJ [[152.95,-29.88,-178.99,-65.32,-58.86,69.58],[9E9,9E9,9E9,9E9,9E9,9E9]],speeddata0,DefaultBlend,tool0;
  MoveAbsJ [[152.54,-29.80,-179.19,-66.31,-58.72,69.27],[9E9,9E9,9E9,9E9,9E9,9E9]],speeddata0,DefaultBlend,tool0;
  MoveAbsJ [[152.13,-29.71,-179.38,-67.30,-58.57,68.96],[9E9,9E9,9E9,9E9,9E9,9E9]],speeddata0,DefaultBlend,tool0;
  MoveAbsJ [[151.72,-29.62,-179.58,-68.29,-58.43,68.65],[9E9,9E9,9E9,9E9,9E9,9E9]],speeddata0,DefaultBlend,tool0;
  MoveAbsJ [[151.31,-29.54,-179.78,-69.28,-58.28,68.34],[9E9,9E9,9E9,9E9,9E9,9E9]],speeddata0,DefaultBlend,tool0;
  MoveAbsJ [[150.90,-29.45,-179.97,-70.27,-58.14,68.03],[9E9,9E9,9E9,9E9,9E9,9E9]],speeddata0,DefaultBlend,tool0;
  MoveAbsJ [[150.49,-29.37,-180.17,-71.26,-57.99,67.72],[9E9,9E9,9E9,9E9,9E9,9E9]],speeddata0,DefaultBlend,tool0;
  MoveAbsJ [[150.08,-29.28,-180.37,-72.25,-57.85,67.41],[9E9,9E9,9E9,9E9,9E9,9E9]],speeddata0,DefaultBlend,tool0;
  MoveAbsJ [[149.67,-29.19,-180.56,-73.24,-57.70,67.10],[9E9,9E9,9E9,9E9,9E9,9E9]],speeddata0,DefaultBlend,tool0;
  MoveAbsJ [[149.26,-29.11,-180.76,-74.23,-57.56,66.79],[9E9,9E9,9E9,9E9,9E9,9E9]],speeddata0,DefaultBlend,tool0;
  MoveAbsJ [[148.85,-29.02,-180.96,-75.22,-57.41,66.48],[9E9,9E9,9E9,9E9,9E9,9E9]],speeddata0,DefaultBlend,tool0;
  MoveAbsJ [[148.44,-28.93,-181.15,-76.21,-57.27,66.17],[9E9,9E9,9E9,9E9,9E9,9E9]],speeddata0,DefaultBlend,tool0;
  MoveAbsJ [[148.03,-28.85,-181.35,-77.20,-57.12,65.86],[9E9,9E9,9E9,9E9,9E9,9E9]],speeddata0,DefaultBlend,tool0;
  MoveAbsJ [[147.62,-28.76,-181.55,-78.19,-56.98,65.55],[9E9,9E9,9E9,9E9,9E9,9E9]],speeddata0,DefaultBlend,tool0;
  MoveAbsJ [[147.21,-28.68,-181.75,-79.18,-56.83,65.24],[9E9,9E9,9E9,9E9,9E9,9E9]],speeddata0,DefaultBlend,tool0;
  MoveAbsJ [[146.80,-28.59,-181.94,-80.17,-56.69,64.93],[9E9,9E9,9E9,9E9,9E9,9E9]],speeddata0,DefaultBlend,tool0;
  MoveAbsJ [[146.39,-28.50,-182.14,-81.16,-56.54,64.62],[9E9,9E9,9E9,9E9,9E9,9E9]],speeddata0,DefaultBlend,tool0;
  MoveAbsJ [[145.98,-28.42,-182.34,-82.15,-56.40,64.31],[9E9,9E9,9E9,9E9,9E9,9E9]],speeddata0,DefaultBlend,tool0;
  MoveAbsJ [[145.58,-28.33,-182.53,-83.14,-56.25,64.01],[9E9,9E9,9E9,9E9,9E9,9E9]],speeddata0,DefaultBlend,tool0;
  MoveAbsJ [[145.17,-28.24,-182.73,-84.13,-56.11,63.70],[9E9,9E9,9E9,9E9,9E9,9E9]],speeddata0,DefaultBlend,tool0;
  MoveAbsJ [[144.76,-28.16,-182.93,-85.12,-55.96,63.39],[9E9,9E9,9E9,9E9,9E9,9E9]],speeddata0,DefaultBlend,tool0;
  MoveAbsJ [[144.35,-28.07,-183.12,-86.11,-55.82,63.08],[9E9,9E9,9E9,9E9,9E9,9E9]],speeddata0,DefaultBlend,tool0;
  MoveAbsJ [[143.94,-27.99,-183.32,-87.10,-55.67,62.77],[9E9,9E9,9E9,9E9,9E9,9E9]],speeddata0,DefaultBlend,tool0;
  MoveAbsJ [[143.53,-27.90,-183.52,-88.09,-55.53,62.46],[9E9,9E9,9E9,9E9,9E9,9E9]],speeddata0,DefaultBlend,tool0;
  MoveAbsJ [[143.12,-27.81,-183.71,-89.08,-55.38,62.15],[9E9,9E9,9E9,9E9,9E9,9E9]],speeddata0,DefaultBlend,tool0;
  MoveAbsJ [[142.71,-27.73,-183.91,-90.07,-55.24,61.84],[9E9,9E9,9E9,9E9,9E9,9E9]],speeddata0,DefaultBlend,tool0;
  MoveAbsJ [[142.30,-27.64,-184.11,-91.06,-55.09,61.53],[9E9,9E9,9E9,9E9,9E9,9E9]],speeddata0,DefaultBlend,tool0;
  MoveAbsJ [[141.89,-27.55,-184.30,-92.05,-54.95,61.22],[9E9,9E9,9E9,9E9,9E9,9E9]],speeddata0,DefaultBlend,tool0;
  MoveAbsJ [[141.48,-27.47,-184.50,-93.04,-54.80,60.91],[9E9,9E9,9E9,9E9,9E9,9E9]],speeddata0,DefaultBlend,tool0;
  MoveAbsJ [[141.07,-27.38,-184.70,-94.03,-54.66,60.60],[9E9,9E9,9E9,9E9,9E9,9E9]],speeddata0,DefaultBlend,tool0;
  MoveAbsJ [[140.66,-27.30,-184.89,-95.02,-54.51,60.29],[9E9,9E9,9E9,9E9,9E9,9E9]],speeddata0,DefaultBlend,tool0;
  MoveAbsJ [[140.25,-27.21,-185.09,-96.01,-54.37,59.98],[9E9,9E9,9E9,9E9,9E9,9E9]],speeddata0,DefaultBlend,tool0;
  MoveAbsJ [[139.84,-27.12,-185.29,-97.00,-54.22,59.67],[9E9,9E9,9E9,9E9,9E9,9E9]],speeddata0,DefaultBlend,tool0;
  MoveAbsJ [[139.43,-27.04,-185.48,-97.99,-54.08,59.36],[9E9,9E9,9E9,9E9,9E9,9E9]],speeddata0,DefaultBlend,tool0;
  MoveAbsJ [[139.02,-26.95,-185.68,-98.98,-53.94,59.05],[9E9,9E9,9E9,9E9,9E9,9E9]],speeddata0,DefaultBlend,tool0;
  MoveAbsJ [[138.61,-26.86,-185.88,-99.97,-53.79,58.74],[9E9,9E9,9E9,9E9,9E9,9E9]],speeddata0,DefaultBlend,tool0;
  MoveAbsJ [[138.20,-26.78,-186.07,-100.96,-53.65,58.44],[9E9,9E9,9E9,9E9,9E9,9E9]],speeddata0,DefaultBlend,tool0;
  MoveAbsJ [[137.79,-26.69,-186.27,-101.95,-53.50,58.13],[9E9,9E9,9E9,9E9,9E9,9E9]],speeddata0,DefaultBlend,tool0;
  MoveAbsJ [[137.38,-26.61,-186.47,-102.93,-53.36,57.82],[9E9,9E9,9E9,9E9,9E9,9E9]],speeddata0,DefaultBlend,tool0;
  MoveAbsJ [[136.97,-26.52,-186.66,-103.92,-53.21,57.51],[9E9,9E9,9E9,9E9,9E9,9E9]],speeddata0,DefaultBlend,tool0;
  MoveAbsJ [[136.56,-26.43,-186.86,-104.91,-53.07,57.20],[9E9,9E9,9E9,9E9,9E9,9E9]],speeddata0,DefaultBlend,tool0;
  MoveAbsJ [[136.15,-26.35,-187.06,-105.90,-52.92,56.89],[9E9,9E9,9E9,9E9,9E9,9E9]],speeddata0,DefaultBlend,tool0;
  MoveAbsJ [[135.74,-26.26,-187.26,-106.89,-52.78,56.58],[9E9,9E9,9E9,9E9,9E9,9E9]],speeddata0,DefaultBlend,tool0;
  MoveAbsJ [[135.33,-26.17,-187.45,-107.88,-52.63,56.27],[9E9,9E9,9E9,9E9,9E9,9E9]],speeddata0,DefaultBlend,tool0;
  MoveAbsJ [[134.92,-26.09,-187.65,-108.87,-52.49,55.96],[9E9,9E9,9E9,9E9,9E9,9E9]],speeddata0,DefaultBlend,tool0;
  MoveAbsJ [[134.51,-26.00,-187.85,-109.86,-52.34,55.65],[9E9,9E9,9E9,9E9,9E9,9E9]],speeddata0,DefaultBlend,tool0;
  MoveAbsJ [[134.10,-25.92,-188.04,-110.85,-52.20,55.34],[9E9,9E9,9E9,9E9,9E9,9E9]],speeddata0,DefaultBlend,tool0;
  MoveAbsJ [[133.69,-25.83,-188.24,-111.84,-52.05,55.03],[9E9,9E9,9E9,9E9,9E9,9E9]],speeddata0,DefaultBlend,tool0;
  MoveAbsJ [[133.28,-25.74,-188.44,-112.83,-51.91,54.72],[9E9,9E9,9E9,9E9,9E9,9E9]],speeddata0,DefaultBlend,tool0;
  MoveAbsJ [[132.87,-25.66,-188.63,-113.82,-51.76,54.41],[9E9,9E9,9E9,9E9,9E9,9E9]],speeddata0,DefaultBlend,tool0;
  MoveAbsJ [[132.46,-25.57,-188.83,-114.81,-51.62,54.10],[9E9,9E9,9E9,9E9,9E9,9E9]],speeddata0,DefaultBlend,tool0;
  MoveAbsJ [[132.05,-25.48,-189.03,-115.80,-51.47,53.79],[9E9,9E9,9E9,9E9,9E9,9E9]],speeddata0,DefaultBlend,tool0;
  MoveAbsJ [[131.64,-25.40,-189.22,-116.79,-51.33,53.48],[9E9,9E9,9E9,9E9,9E9,9E9]],speeddata0,DefaultBlend,tool0;
  MoveAbsJ [[131.23,-25.31,-189.42,-117.78,-51.18,53.17],[9E9,9E9,9E9,9E9,9E9,9E9]],speeddata0,DefaultBlend,tool0;
  MoveAbsJ [[130.82,-25.23,-189.62,-118.77,-51.04,52.87],[9E9,9E9,9E9,9E9,9E9,9E9]],speeddata0,DefaultBlend,tool0;
  MoveAbsJ [[130.41,-25.14,-189.81,-119.76,-50.89,52.56],[9E9,9E9,9E9,9E9,9E9,9E9]],speeddata0,DefaultBlend,tool0;
  MoveAbsJ [[130.00,-25.05,-190.01,-120.75,-50.75,52.25],[9E9,9E9,9E9,9E9,9E9,9E9]],speeddata0,DefaultBlend,tool0;
  MoveAbsJ [[129.59,-24.97,-190.21,-121.74,-50.60,51.94],[9E9,9E9,9E9,9E9,9E9,9E9]],speeddata0,DefaultBlend,tool0;
  MoveAbsJ [[129.18,-24.88,-190.40,-122.73,-50.46,51.63],[9E9,9E9,9E9,9E9,9E9,9E9]],speeddata0,DefaultBlend,tool0;
  MoveAbsJ [[128.77,-24.79,-190.60,-123.72,-50.31,51.32],[9E9,9E9,9E9,9E9,9E9,9E9]],speeddata0,DefaultBlend,tool0;
  MoveAbsJ [[128.36,-24.71,-190.80,-124.71,-50.17,51.01],[9E9,9E9,9E9,9E9,9E9,9E9]],speeddata0,DefaultBlend,tool0;
  MoveAbsJ [[127.95,-24.62,-190.99,-125.70,-50.02,50.70],[9E9,9E9,9E9,9E9,9E9,9E9]],speeddata0,DefaultBlend,tool0;
  MoveAbsJ [[127.54,-24.54,-191.19,-126.69,-49.88,50.39],[9E9,9E9,9E9,9E9,9E9,9E9]],speeddata0,DefaultBlend,tool0;
  MoveAbsJ [[127.13,-24.45,-191.39,-127.68,-49.73,50.08],[9E9,9E9,9E9,9E9,9E9,9E9]],speeddata0,FinePoint,tool0;
  TPWrite "Action 22 LoadWorkpiece.";
  TPWrite "Press Play to Continue";
  Stop;
  TPWrite "Action 23 CloseGripper.";
  TPWrite "Press Play to Continue";
  Stop;
  TPWrite "Action 24 FreeMovement.";
  MoveAbsJ [[127.13,-24.45,-191.39,-127.68,-49.73,50.08],[9E9,9E9,9E9,9E9,9E9,9E9]],speeddata0,DefaultBlend,tool0;
  MoveAbsJ [[126.87,-24.11,-191.00,-127.69,-49.49,49.58],[9E9,9E9,9E9,9E9,9E9,9E9]],speeddata0,DefaultBlend,tool0;
  MoveAbsJ [[126.65,-23.69,-190.02,-127.13,-49.25,48.92],[9E9,9E9,9E9,9E9,9E9,9E9]],speeddata0,DefaultBlend,tool0;
  MoveAbsJ [[126.94,-23.83,-189.31,-126.15,-49.43,49.02],[9E9,9E9,9E9,9E9,9E9,9E9]],speeddata0,DefaultBlend,tool0;
  MoveAbsJ [[127.23,-23.96,-188.61,-125.17,-49.62,49.11],[9E9,9E9,9E9,9E9,9E9,9E9]],speeddata0,DefaultBlend,tool0;
  MoveAbsJ [[127.53,-24.10,-187.90,-124.19,-49.81,49.21],[9E9,9E9,9E9,9E9,9E9,9E9]],speeddata0,DefaultBlend,tool0;
  MoveAbsJ [[127.82,-24.24,-187.19,-123.21,-50.00,49.30],[9E9,9E9,9E9,9E9,9E9,9E9]],speeddata0,DefaultBlend,tool0;
  MoveAbsJ [[128.11,-24.38,-186.48,-122.23,-50.19,49.40],[9E9,9E9,9E9,9E9,9E9,9E9]],speeddata0,DefaultBlend,tool0;
  MoveAbsJ [[128.41,-24.51,-185.78,-121.26,-50.38,49.50],[9E9,9E9,9E9,9E9,9E9,9E9]],speeddata0,DefaultBlend,tool0;
  MoveAbsJ [[128.70,-24.65,-185.07,-120.28,-50.57,49.59],[9E9,9E9,9E9,9E9,9E9,9E9]],speeddata0,DefaultBlend,tool0;
  MoveAbsJ [[128.99,-24.79,-184.36,-119.30,-50.76,49.69],[9E9,9E9,9E9,9E9,9E9,9E9]],speeddata0,DefaultBlend,tool0;
  MoveAbsJ [[129.28,-24.93,-183.65,-118.32,-50.95,49.78],[9E9,9E9,9E9,9E9,9E9,9E9]],speeddata0,DefaultBlend,tool0;
  MoveAbsJ [[129.58,-25.06,-182.95,-117.34,-51.14,49.88],[9E9,9E9,9E9,9E9,9E9,9E9]],speeddata0,DefaultBlend,tool0;
  MoveAbsJ [[129.87,-25.20,-182.24,-116.36,-51.33,49.98],[9E9,9E9,9E9,9E9,9E9,9E9]],speeddata0,DefaultBlend,tool0;
  MoveAbsJ [[130.16,-25.34,-181.53,-115.38,-51.51,50.07],[9E9,9E9,9E9,9E9,9E9,9E9]],speeddata0,DefaultBlend,tool0;
  MoveAbsJ [[130.46,-25.47,-180.82,-114.40,-51.70,50.17],[9E9,9E9,9E9,9E9,9E9,9E9]],speeddata0,DefaultBlend,tool0;
  MoveAbsJ [[130.75,-25.61,-180.12,-113.43,-51.89,50.26],[9E9,9E9,9E9,9E9,9E9,9E9]],speeddata0,DefaultBlend,tool0;
  MoveAbsJ [[131.04,-25.75,-179.41,-112.45,-52.08,50.36],[9E9,9E9,9E9,9E9,9E9,9E9]],speeddata0,DefaultBlend,tool0;
  MoveAbsJ [[131.33,-25.89,-178.70,-111.47,-52.27,50.46],[9E9,9E9,9E9,9E9,9E9,9E9]],speeddata0,DefaultBlend,tool0;
  MoveAbsJ [[131.63,-26.02,-177.99,-110.49,-52.46,50.55],[9E9,9E9,9E9,9E9,9E9,9E9]],speeddata0,DefaultBlend,tool0;
  MoveAbsJ [[131.92,-26.16,-177.29,-109.51,-52.65,50.65],[9E9,9E9,9E9,9E9,9E9,9E9]],speeddata0,DefaultBlend,tool0;
  MoveAbsJ [[132.21,-26.30,-176.58,-108.53,-52.84,50.74],[9E9,9E9,9E9,9E9,9E9,9E9]],speeddata0,DefaultBlend,tool0;
  MoveAbsJ [[132.51,-26.44,-175.87,-107.55,-53.03,50.84],[9E9,9E9,9E9,9E9,9E9,9E9]],speeddata0,DefaultBlend,tool0;
  MoveAbsJ [[132.80,-26.57,-175.16,-106.58,-53.22,50.94],[9E9,9E9,9E9,9E9,9E9,9E9]],speeddata0,DefaultBlend,tool0;
  MoveAbsJ [[133.09,-26.71,-174.46,-105.60,-53.41,51.03],[9E9,9E9,9E9,9E9,9E9,9E9]],speeddata0,DefaultBlend,tool0;
  MoveAbsJ [[133.38,-26.85,-173.75,-104.62,-53.60,51.13],[9E9,9E9,9E9,9E9,9E9,9E9]],speeddata0,DefaultBlend,tool0;
  MoveAbsJ [[133.68,-26.99,-173.04,-103.64,-53.78,51.22],[9E9,9E9,9E9,9E9,9E9,9E9]],speeddata0,DefaultBlend,tool0;
  MoveAbsJ [[133.97,-27.12,-172.34,-102.66,-53.97,51.32],[9E9,9E9,9E9,9E9,9E9,9E9]],speeddata0,DefaultBlend,tool0;
  MoveAbsJ [[134.26,-27.26,-171.63,-101.68,-54.16,51.42],[9E9,9E9,9E9,9E9,9E9,9E9]],speeddata0,DefaultBlend,tool0;
  MoveAbsJ [[134.56,-27.40,-170.92,-100.70,-54.35,51.51],[9E9,9E9,9E9,9E9,9E9,9E9]],speeddata0,DefaultBlend,tool0;
  MoveAbsJ [[134.85,-27.53,-170.21,-99.72,-54.54,51.61],[9E9,9E9,9E9,9E9,9E9,9E9]],speeddata0,DefaultBlend,tool0;
  MoveAbsJ [[135.14,-27.67,-169.51,-98.75,-54.73,51.70],[9E9,9E9,9E9,9E9,9E9,9E9]],speeddata0,DefaultBlend,tool0;
  MoveAbsJ [[135.43,-27.81,-168.80,-97.77,-54.92,51.80],[9E9,9E9,9E9,9E9,9E9,9E9]],speeddata0,DefaultBlend,tool0;
  MoveAbsJ [[135.73,-27.95,-168.09,-96.79,-55.11,51.90],[9E9,9E9,9E9,9E9,9E9,9E9]],speeddata0,DefaultBlend,tool0;
  MoveAbsJ [[136.02,-28.08,-167.38,-95.81,-55.30,51.99],[9E9,9E9,9E9,9E9,9E9,9E9]],speeddata0,DefaultBlend,tool0;
  MoveAbsJ [[136.31,-28.22,-166.68,-94.83,-55.49,52.09],[9E9,9E9,9E9,9E9,9E9,9E9]],speeddata0,DefaultBlend,tool0;
  MoveAbsJ [[136.61,-28.36,-165.97,-93.85,-55.68,52.18],[9E9,9E9,9E9,9E9,9E9,9E9]],speeddata0,DefaultBlend,tool0;
  MoveAbsJ [[136.90,-28.50,-165.26,-92.87,-55.86,52.28],[9E9,9E9,9E9,9E9,9E9,9E9]],speeddata0,DefaultBlend,tool0;
  MoveAbsJ [[137.19,-28.63,-164.55,-91.90,-56.05,52.38],[9E9,9E9,9E9,9E9,9E9,9E9]],speeddata0,DefaultBlend,tool0;
  MoveAbsJ [[137.48,-28.77,-163.85,-90.92,-56.24,52.47],[9E9,9E9,9E9,9E9,9E9,9E9]],speeddata0,DefaultBlend,tool0;
  MoveAbsJ [[137.78,-28.91,-163.14,-89.94,-56.43,52.57],[9E9,9E9,9E9,9E9,9E9,9E9]],speeddata0,DefaultBlend,tool0;
  MoveAbsJ [[138.07,-29.04,-162.43,-88.96,-56.62,52.66],[9E9,9E9,9E9,9E9,9E9,9E9]],speeddata0,DefaultBlend,tool0;
  MoveAbsJ [[138.36,-29.18,-161.72,-87.98,-56.81,52.76],[9E9,9E9,9E9,9E9,9E9,9E9]],speeddata0,DefaultBlend,tool0;
  MoveAbsJ [[138.66,-29.32,-161.02,-87.00,-57.00,52.86],[9E9,9E9,9E9,9E9,9E9,9E9]],speeddata0,DefaultBlend,tool0;
  MoveAbsJ [[138.95,-29.46,-160.31,-86.02,-57.19,52.95],[9E9,9E9,9E9,9E9,9E9,9E9]],speeddata0,DefaultBlend,tool0;
  MoveAbsJ [[139.24,-29.59,-159.60,-85.04,-57.38,53.05],[9E9,9E9,9E9,9E9,9E9,9E9]],speeddata0,DefaultBlend,tool0;
  MoveAbsJ [[139.53,-29.73,-158.89,-84.07,-57.57,53.14],[9E9,9E9,9E9,9E9,9E9,9E9]],speeddata0,DefaultBlend,tool0;
  MoveAbsJ [[139.83,-29.87,-158.19,-83.09,-57.76,53.24],[9E9,9E9,9E9,9E9,9E9,9E9]],speeddata0,DefaultBlend,tool0;
  MoveAbsJ [[140.12,-30.01,-157.48,-82.11,-57.94,53.34],[9E9,9E9,9E9,9E9,9E9,9E9]],speeddata0,DefaultBlend,tool0;
  MoveAbsJ [[140.41,-30.14,-156.77,-81.13,-58.13,53.43],[9E9,9E9,9E9,9E9,9E9,9E9]],speeddata0,DefaultBlend,tool0;
  MoveAbsJ [[140.71,-30.28,-156.06,-80.15,-58.32,53.53],[9E9,9E9,9E9,9E9,9E9,9E9]],speeddata0,DefaultBlend,tool0;
  MoveAbsJ [[141.00,-30.42,-155.36,-79.17,-58.51,53.62],[9E9,9E9,9E9,9E9,9E9,9E9]],speeddata0,DefaultBlend,tool0;
  MoveAbsJ [[141.29,-30.56,-154.65,-78.19,-58.70,53.72],[9E9,9E9,9E9,9E9,9E9,9E9]],speeddata0,DefaultBlend,tool0;
  MoveAbsJ [[141.58,-30.69,-153.94,-77.21,-58.89,53.82],[9E9,9E9,9E9,9E9,9E9,9E9]],speeddata0,DefaultBlend,tool0;
  MoveAbsJ [[141.88,-30.83,-153.23,-76.24,-59.08,53.91],[9E9,9E9,9E9,9E9,9E9,9E9]],speeddata0,DefaultBlend,tool0;
  MoveAbsJ [[142.17,-30.97,-152.53,-75.26,-59.27,54.01],[9E9,9E9,9E9,9E9,9E9,9E9]],speeddata0,DefaultBlend,tool0;
  MoveAbsJ [[142.46,-31.10,-151.82,-74.28,-59.46,54.10],[9E9,9E9,9E9,9E9,9E9,9E9]],speeddata0,DefaultBlend,tool0;
  MoveAbsJ [[142.76,-31.24,-151.11,-73.30,-59.65,54.20],[9E9,9E9,9E9,9E9,9E9,9E9]],speeddata0,DefaultBlend,tool0;
  MoveAbsJ [[143.05,-31.38,-150.40,-72.32,-59.84,54.30],[9E9,9E9,9E9,9E9,9E9,9E9]],speeddata0,DefaultBlend,tool0;
  MoveAbsJ [[143.34,-31.52,-149.70,-71.34,-60.02,54.39],[9E9,9E9,9E9,9E9,9E9,9E9]],speeddata0,DefaultBlend,tool0;
  MoveAbsJ [[143.63,-31.65,-148.99,-70.36,-60.21,54.49],[9E9,9E9,9E9,9E9,9E9,9E9]],speeddata0,DefaultBlend,tool0;
  MoveAbsJ [[143.93,-31.79,-148.28,-69.39,-60.40,54.58],[9E9,9E9,9E9,9E9,9E9,9E9]],speeddata0,DefaultBlend,tool0;
  MoveAbsJ [[144.22,-31.93,-147.57,-68.41,-60.59,54.68],[9E9,9E9,9E9,9E9,9E9,9E9]],speeddata0,DefaultBlend,tool0;
  MoveAbsJ [[144.51,-32.07,-146.87,-67.43,-60.78,54.78],[9E9,9E9,9E9,9E9,9E9,9E9]],speeddata0,DefaultBlend,tool0;
  MoveAbsJ [[144.81,-32.20,-146.16,-66.45,-60.97,54.87],[9E9,9E9,9E9,9E9,9E9,9E9]],speeddata0,DefaultBlend,tool0;
  MoveAbsJ [[145.10,-32.34,-145.45,-65.47,-61.16,54.97],[9E9,9E9,9E9,9E9,9E9,9E9]],speeddata0,DefaultBlend,tool0;
  MoveAbsJ [[145.39,-32.48,-144.74,-64.49,-61.35,55.06],[9E9,9E9,9E9,9E9,9E9,9E9]],speeddata0,DefaultBlend,tool0;
  MoveAbsJ [[145.68,-32.61,-144.04,-63.51,-61.54,55.16],[9E9,9E9,9E9,9E9,9E9,9E9]],speeddata0,DefaultBlend,tool0;
  MoveAbsJ [[145.98,-32.75,-143.33,-62.53,-61.73,55.26],[9E9,9E9,9E9,9E9,9E9,9E9]],speeddata0,DefaultBlend,tool0;
  MoveAbsJ [[146.27,-32.89,-142.62,-61.56,-61.92,55.35],[9E9,9E9,9E9,9E9,9E9,9E9]],speeddata0,DefaultBlend,tool0;
  MoveAbsJ [[146.56,-33.03,-141.91,-60.58,-62.11,55.45],[9E9,9E9,9E9,9E9,9E9,9E9]],speeddata0,DefaultBlend,tool0;
  MoveAbsJ [[146.85,-33.16,-141.21,-59.60,-62.29,55.54],[9E9,9E9,9E9,9E9,9E9,9E9]],speeddata0,DefaultBlend,tool0;
  MoveAbsJ [[147.15,-33.30,-140.50,-58.62,-62.48,55.64],[9E9,9E9,9E9,9E9,9E9,9E9]],speeddata0,DefaultBlend,tool0;
  MoveAbsJ [[147.44,-33.44,-139.79,-57.64,-62.67,55.74],[9E9,9E9,9E9,9E9,9E9,9E9]],speeddata0,DefaultBlend,tool0;
  MoveAbsJ [[147.73,-33.58,-139.08,-56.66,-62.86,55.83],[9E9,9E9,9E9,9E9,9E9,9E9]],speeddata0,DefaultBlend,tool0;
  MoveAbsJ [[148.03,-33.71,-138.38,-55.68,-63.05,55.93],[9E9,9E9,9E9,9E9,9E9,9E9]],speeddata0,DefaultBlend,tool0;
  MoveAbsJ [[148.32,-33.85,-137.67,-54.70,-63.24,56.02],[9E9,9E9,9E9,9E9,9E9,9E9]],speeddata0,DefaultBlend,tool0;
  MoveAbsJ [[148.61,-33.99,-136.96,-53.73,-63.43,56.12],[9E9,9E9,9E9,9E9,9E9,9E9]],speeddata0,DefaultBlend,tool0;
  MoveAbsJ [[148.90,-34.12,-136.25,-52.75,-63.62,56.22],[9E9,9E9,9E9,9E9,9E9,9E9]],speeddata0,DefaultBlend,tool0;
  MoveAbsJ [[149.20,-34.26,-135.55,-51.77,-63.81,56.31],[9E9,9E9,9E9,9E9,9E9,9E9]],speeddata0,DefaultBlend,tool0;
  MoveAbsJ [[149.49,-34.40,-134.84,-50.79,-64.00,56.41],[9E9,9E9,9E9,9E9,9E9,9E9]],speeddata0,DefaultBlend,tool0;
  MoveAbsJ [[149.78,-34.54,-134.13,-49.81,-64.19,56.50],[9E9,9E9,9E9,9E9,9E9,9E9]],speeddata0,DefaultBlend,tool0;
  MoveAbsJ [[150.08,-34.67,-133.42,-48.83,-64.37,56.60],[9E9,9E9,9E9,9E9,9E9,9E9]],speeddata0,DefaultBlend,tool0;
  MoveAbsJ [[150.37,-34.81,-132.72,-47.85,-64.56,56.70],[9E9,9E9,9E9,9E9,9E9,9E9]],speeddata0,DefaultBlend,tool0;
  MoveAbsJ [[150.66,-34.95,-132.01,-46.88,-64.75,56.79],[9E9,9E9,9E9,9E9,9E9,9E9]],speeddata0,DefaultBlend,tool0;
  MoveAbsJ [[150.95,-35.09,-131.30,-45.90,-64.94,56.89],[9E9,9E9,9E9,9E9,9E9,9E9]],speeddata0,DefaultBlend,tool0;
  MoveAbsJ [[151.25,-35.22,-130.59,-44.92,-65.13,56.98],[9E9,9E9,9E9,9E9,9E9,9E9]],speeddata0,DefaultBlend,tool0;
  MoveAbsJ [[151.54,-35.36,-129.89,-43.94,-65.32,57.08],[9E9,9E9,9E9,9E9,9E9,9E9]],speeddata0,DefaultBlend,tool0;
  MoveAbsJ [[151.83,-35.50,-129.18,-42.96,-65.51,57.18],[9E9,9E9,9E9,9E9,9E9,9E9]],speeddata0,DefaultBlend,tool0;
  MoveAbsJ [[152.00,-35.59,-128.85,-42.47,-65.62,57.26],[9E9,9E9,9E9,9E9,9E9,9E9]],speeddata0,DefaultBlend,tool0;
  MoveAbsJ [[152.34,-35.78,-128.20,-41.48,-65.85,57.43],[9E9,9E9,9E9,9E9,9E9,9E9]],speeddata0,DefaultBlend,tool0;
  MoveAbsJ [[152.67,-35.97,-127.55,-40.50,-66.08,57.61],[9E9,9E9,9E9,9E9,9E9,9E9]],speeddata0,DefaultBlend,tool0;
  MoveAbsJ [[153.01,-36.17,-126.90,-39.51,-66.31,57.78],[9E9,9E9,9E9,9E9,9E9,9E9]],speeddata0,DefaultBlend,tool0;
  MoveAbsJ [[153.34,-36.36,-126.24,-38.52,-66.53,57.95],[9E9,9E9,9E9,9E9,9E9,9E9]],speeddata0,DefaultBlend,tool0;
  MoveAbsJ [[153.68,-36.55,-125.59,-37.54,-66.76,58.13],[9E9,9E9,9E9,9E9,9E9,9E9]],speeddata0,DefaultBlend,tool0;
  MoveAbsJ [[154.02,-36.74,-124.94,-36.55,-66.99,58.30],[9E9,9E9,9E9,9E9,9E9,9E9]],speeddata0,DefaultBlend,tool0;
  MoveAbsJ [[154.72,-37.40,-124.83,-35.56,-67.55,59.15],[9E9,9E9,9E9,9E9,9E9,9E9]],speeddata0,DefaultBlend,tool0;
  MoveAbsJ [[155.42,-38.06,-124.72,-34.58,-68.12,60.01],[9E9,9E9,9E9,9E9,9E9,9E9]],speeddata0,DefaultBlend,tool0;
  MoveAbsJ [[156.12,-38.72,-124.61,-33.59,-68.68,60.87],[9E9,9E9,9E9,9E9,9E9,9E9]],speeddata0,DefaultBlend,tool0;
  MoveAbsJ [[156.83,-39.39,-124.50,-32.60,-69.24,61.73],[9E9,9E9,9E9,9E9,9E9,9E9]],speeddata0,DefaultBlend,tool0;
  MoveAbsJ [[157.53,-40.05,-124.40,-31.61,-69.81,62.58],[9E9,9E9,9E9,9E9,9E9,9E9]],speeddata0,DefaultBlend,tool0;
  MoveAbsJ [[158.23,-40.71,-124.29,-30.62,-70.37,63.44],[9E9,9E9,9E9,9E9,9E9,9E9]],speeddata0,DefaultBlend,tool0;
  MoveAbsJ [[158.93,-41.37,-124.18,-29.64,-70.93,64.30],[9E9,9E9,9E9,9E9,9E9,9E9]],speeddata0,DefaultBlend,tool0;
  MoveAbsJ [[159.63,-42.04,-124.07,-28.65,-71.50,65.15],[9E9,9E9,9E9,9E9,9E9,9E9]],speeddata0,DefaultBlend,tool0;
  MoveAbsJ [[160.34,-42.70,-123.96,-27.66,-72.06,66.01],[9E9,9E9,9E9,9E9,9E9,9E9]],speeddata0,DefaultBlend,tool0;
  MoveAbsJ [[161.04,-43.36,-123.85,-26.67,-72.62,66.87],[9E9,9E9,9E9,9E9,9E9,9E9]],speeddata0,DefaultBlend,tool0;
  MoveAbsJ [[161.74,-44.02,-123.74,-25.68,-73.19,67.72],[9E9,9E9,9E9,9E9,9E9,9E9]],speeddata0,DefaultBlend,tool0;
  MoveAbsJ [[162.44,-44.68,-123.64,-24.70,-73.75,68.58],[9E9,9E9,9E9,9E9,9E9,9E9]],speeddata0,DefaultBlend,tool0;
  MoveAbsJ [[163.15,-45.35,-123.53,-23.71,-74.31,69.44],[9E9,9E9,9E9,9E9,9E9,9E9]],speeddata0,DefaultBlend,tool0;
  MoveAbsJ [[163.85,-46.01,-123.42,-22.72,-74.88,70.29],[9E9,9E9,9E9,9E9,9E9,9E9]],speeddata0,DefaultBlend,tool0;
  MoveAbsJ [[164.55,-46.67,-123.31,-21.73,-75.44,71.15],[9E9,9E9,9E9,9E9,9E9,9E9]],speeddata0,DefaultBlend,tool0;
  MoveAbsJ [[165.25,-47.33,-123.20,-20.75,-76.00,72.01],[9E9,9E9,9E9,9E9,9E9,9E9]],speeddata0,DefaultBlend,tool0;
  MoveAbsJ [[165.95,-48.00,-123.09,-19.76,-76.57,72.86],[9E9,9E9,9E9,9E9,9E9,9E9]],speeddata0,DefaultBlend,tool0;
  MoveAbsJ [[166.66,-48.66,-122.98,-18.77,-77.13,73.72],[9E9,9E9,9E9,9E9,9E9,9E9]],speeddata0,DefaultBlend,tool0;
  MoveAbsJ [[167.36,-49.32,-122.88,-17.78,-77.70,74.58],[9E9,9E9,9E9,9E9,9E9,9E9]],speeddata0,DefaultBlend,tool0;
  MoveAbsJ [[168.06,-49.98,-122.77,-16.79,-78.26,75.43],[9E9,9E9,9E9,9E9,9E9,9E9]],speeddata0,DefaultBlend,tool0;
  MoveAbsJ [[168.76,-50.64,-122.66,-15.81,-78.82,76.29],[9E9,9E9,9E9,9E9,9E9,9E9]],speeddata0,DefaultBlend,tool0;
  MoveAbsJ [[169.47,-51.31,-122.55,-14.82,-79.39,77.15],[9E9,9E9,9E9,9E9,9E9,9E9]],speeddata0,DefaultBlend,tool0;
  MoveAbsJ [[170.17,-51.97,-122.44,-13.83,-79.95,78.00],[9E9,9E9,9E9,9E9,9E9,9E9]],speeddata0,DefaultBlend,tool0;
  MoveAbsJ [[170.87,-52.63,-122.33,-12.84,-80.51,78.86],[9E9,9E9,9E9,9E9,9E9,9E9]],speeddata0,DefaultBlend,tool0;
  MoveAbsJ [[171.57,-53.29,-122.22,-11.85,-81.08,79.72],[9E9,9E9,9E9,9E9,9E9,9E9]],speeddata0,DefaultBlend,tool0;
  MoveAbsJ [[172.28,-53.96,-122.12,-10.87,-81.64,80.58],[9E9,9E9,9E9,9E9,9E9,9E9]],speeddata0,DefaultBlend,tool0;
  MoveAbsJ [[172.98,-54.62,-122.01,-9.88,-82.20,81.43],[9E9,9E9,9E9,9E9,9E9,9E9]],speeddata0,DefaultBlend,tool0;
  MoveAbsJ [[173.68,-55.28,-121.90,-8.89,-82.77,82.29],[9E9,9E9,9E9,9E9,9E9,9E9]],speeddata0,DefaultBlend,tool0;
  MoveAbsJ [[174.38,-55.94,-121.79,-7.90,-83.33,83.15],[9E9,9E9,9E9,9E9,9E9,9E9]],speeddata0,DefaultBlend,tool0;
  MoveAbsJ [[175.08,-56.60,-121.68,-6.92,-83.89,84.00],[9E9,9E9,9E9,9E9,9E9,9E9]],speeddata0,DefaultBlend,tool0;
  MoveAbsJ [[175.79,-57.27,-121.57,-5.93,-84.46,84.86],[9E9,9E9,9E9,9E9,9E9,9E9]],speeddata0,DefaultBlend,tool0;
  MoveAbsJ [[176.49,-57.93,-121.46,-4.94,-85.02,85.72],[9E9,9E9,9E9,9E9,9E9,9E9]],speeddata0,DefaultBlend,tool0;
  MoveAbsJ [[177.19,-58.59,-121.36,-3.95,-85.58,86.57],[9E9,9E9,9E9,9E9,9E9,9E9]],speeddata0,DefaultBlend,tool0;
  MoveAbsJ [[177.89,-59.25,-121.25,-2.96,-86.15,87.43],[9E9,9E9,9E9,9E9,9E9,9E9]],speeddata0,DefaultBlend,tool0;
  MoveAbsJ [[178.60,-59.92,-121.14,-1.98,-86.71,88.29],[9E9,9E9,9E9,9E9,9E9,9E9]],speeddata0,DefaultBlend,tool0;
  MoveAbsJ [[179.30,-60.58,-121.03,-0.99,-87.27,89.14],[9E9,9E9,9E9,9E9,9E9,9E9]],speeddata0,DefaultBlend,tool0;
  MoveAbsJ [[180.00,-61.24,-120.92,0.00,-87.84,90.00],[9E9,9E9,9E9,9E9,9E9,9E9]],speeddata0,FinePoint,tool0;
  TPWrite "Action 25 LinearMovement.";
  MoveAbsJ [[180.00,-61.24,-120.92,0.00,-87.84,90.00],[9E9,9E9,9E9,9E9,9E9,9E9]],speeddata0,DefaultBlend,tool0;
  MoveAbsJ [[180.00,-61.80,-121.04,0.00,-87.16,90.00],[9E9,9E9,9E9,9E9,9E9,9E9]],speeddata0,DefaultBlend,tool0;
  MoveAbsJ [[180.00,-62.32,-121.24,0.00,-86.45,90.00],[9E9,9E9,9E9,9E9,9E9,9E9]],speeddata0,DefaultBlend,tool0;
  MoveAbsJ [[180.00,-62.84,-121.45,0.00,-85.72,90.00],[9E9,9E9,9E9,9E9,9E9,9E9]],speeddata0,DefaultBlend,tool0;
  MoveAbsJ [[180.00,-63.36,-121.65,0.00,-85.00,90.00],[9E9,9E9,9E9,9E9,9E9,9E9]],speeddata0,DefaultBlend,tool0;
  MoveAbsJ [[180.00,-63.89,-121.82,0.00,-84.29,90.00],[9E9,9E9,9E9,9E9,9E9,9E9]],speeddata0,DefaultBlend,tool0;
  MoveAbsJ [[180.00,-64.44,-121.97,0.00,-83.59,90.00],[9E9,9E9,9E9,9E9,9E9,9E9]],speeddata0,DefaultBlend,tool0;
  MoveAbsJ [[180.00,-65.01,-122.08,0.00,-82.91,90.00],[9E9,9E9,9E9,9E9,9E9,9E9]],speeddata0,DefaultBlend,tool0;
  MoveAbsJ [[180.00,-65.60,-122.16,0.00,-82.24,90.00],[9E9,9E9,9E9,9E9,9E9,9E9]],speeddata0,FinePoint,tool0;
  TPWrite "Action 26 OpenGripper.";
  TPWrite "Press Play to Continue";
  Stop;
  TPWrite "Action 27 LinearMovement.";
  MoveAbsJ [[180.00,-65.58,-122.19,0.00,-82.23,90.00],[9E9,9E9,9E9,9E9,9E9,9E9]],speeddata0,DefaultBlend,tool0;
  MoveAbsJ [[180.00,-64.97,-122.17,0.00,-82.86,90.00],[9E9,9E9,9E9,9E9,9E9,9E9]],speeddata0,DefaultBlend,tool0;
  MoveAbsJ [[180.00,-64.37,-122.11,0.00,-83.52,90.00],[9E9,9E9,9E9,9E9,9E9,9E9]],speeddata0,DefaultBlend,tool0;
  MoveAbsJ [[180.00,-63.79,-122.02,0.00,-84.19,90.00],[9E9,9E9,9E9,9E9,9E9,9E9]],speeddata0,DefaultBlend,tool0;
  MoveAbsJ [[180.00,-63.23,-121.89,0.00,-84.88,90.00],[9E9,9E9,9E9,9E9,9E9,9E9]],speeddata0,DefaultBlend,tool0;
  MoveAbsJ [[180.00,-62.69,-121.73,0.00,-85.58,90.00],[9E9,9E9,9E9,9E9,9E9,9E9]],speeddata0,DefaultBlend,tool0;
  MoveAbsJ [[180.00,-62.16,-121.54,0.00,-86.30,90.00],[9E9,9E9,9E9,9E9,9E9,9E9]],speeddata0,DefaultBlend,tool0;
  MoveAbsJ [[180.00,-61.66,-121.31,0.00,-87.03,90.00],[9E9,9E9,9E9,9E9,9E9,9E9]],speeddata0,DefaultBlend,tool0;
  MoveAbsJ [[180.00,-61.17,-121.05,0.00,-87.77,90.00],[9E9,9E9,9E9,9E9,9E9,9E9]],speeddata0,FinePoint,tool0;
  TPWrite "Action 28 FreeMovement.";
  MoveAbsJ [[180.00,-61.17,-121.05,0.00,-87.77,90.00],[9E9,9E9,9E9,9E9,9E9,9E9]],speeddata0,DefaultBlend,tool0;
  MoveAbsJ [[179.59,-60.89,-121.59,-0.99,-87.48,89.69],[9E9,9E9,9E9,9E9,9E9,9E9]],speeddata0,DefaultBlend,tool0;
  MoveAbsJ [[179.18,-60.60,-122.14,-1.98,-87.18,89.38],[9E9,9E9,9E9,9E9,9E9,9E9]],speeddata0,DefaultBlend,tool0;
  MoveAbsJ [[178.77,-60.32,-122.69,-2.97,-86.89,89.07],[9E9,9E9,9E9,9E9,9E9,9E9]],speeddata0,DefaultBlend,tool0;
  MoveAbsJ [[178.36,-60.03,-123.23,-3.96,-86.59,88.76],[9E9,9E9,9E9,9E9,9E9,9E9]],speeddata0,DefaultBlend,tool0;
  MoveAbsJ [[177.95,-59.75,-123.78,-4.95,-86.30,88.46],[9E9,9E9,9E9,9E9,9E9,9E9]],speeddata0,DefaultBlend,tool0;
  MoveAbsJ [[177.54,-59.47,-124.32,-5.94,-86.00,88.15],[9E9,9E9,9E9,9E9,9E9,9E9]],speeddata0,DefaultBlend,tool0;
  MoveAbsJ [[177.13,-59.18,-124.87,-6.93,-85.71,87.84],[9E9,9E9,9E9,9E9,9E9,9E9]],speeddata0,DefaultBlend,tool0;
  MoveAbsJ [[176.72,-58.90,-125.41,-7.92,-85.41,87.53],[9E9,9E9,9E9,9E9,9E9,9E9]],speeddata0,DefaultBlend,tool0;
  MoveAbsJ [[176.31,-58.61,-125.96,-8.91,-85.12,87.22],[9E9,9E9,9E9,9E9,9E9,9E9]],speeddata0,DefaultBlend,tool0;
  MoveAbsJ [[175.90,-58.33,-126.50,-9.90,-84.82,86.91],[9E9,9E9,9E9,9E9,9E9,9E9]],speeddata0,DefaultBlend,tool0;
  MoveAbsJ [[175.49,-58.04,-127.05,-10.89,-84.53,86.60],[9E9,9E9,9E9,9E9,9E9,9E9]],speeddata0,DefaultBlend,tool0;
  MoveAbsJ [[175.08,-57.76,-127.59,-11.88,-84.24,86.29],[9E9,9E9,9E9,9E9,9E9,9E9]],speeddata0,DefaultBlend,tool0;
  MoveAbsJ [[174.67,-57.47,-128.14,-12.87,-83.94,85.98],[9E9,9E9,9E9,9E9,9E9,9E9]],speeddata0,DefaultBlend,tool0;
  MoveAbsJ [[174.26,-57.19,-128.69,-13.86,-83.65,85.67],[9E9,9E9,9E9,9E9,9E9,9E9]],speeddata0,DefaultBlend,tool0;
  MoveAbsJ [[173.85,-56.90,-129.23,-14.85,-83.35,85.37],[9E9,9E9,9E9,9E9,9E9,9E9]],speeddata0,DefaultBlend,tool0;
  MoveAbsJ [[173.44,-56.62,-129.78,-15.84,-83.06,85.06],[9E9,9E9,9E9,9E9,9E9,9E9]],speeddata0,DefaultBlend,tool0;
  MoveAbsJ [[173.03,-56.34,-130.32,-16.83,-82.76,84.75],[9E9,9E9,9E9,9E9,9E9,9E9]],speeddata0,DefaultBlend,tool0;
  MoveAbsJ [[172.62,-56.05,-130.87,-17.82,-82.47,84.44],[9E9,9E9,9E9,9E9,9E9,9E9]],speeddata0,DefaultBlend,tool0;
  MoveAbsJ [[172.21,-55.77,-131.41,-18.81,-82.17,84.13],[9E9,9E9,9E9,9E9,9E9,9E9]],speeddata0,DefaultBlend,tool0;
  MoveAbsJ [[171.80,-55.48,-131.96,-19.81,-81.88,83.82],[9E9,9E9,9E9,9E9,9E9,9E9]],speeddata0,DefaultBlend,tool0;
  MoveAbsJ [[171.39,-55.20,-132.50,-20.80,-81.58,83.51],[9E9,9E9,9E9,9E9,9E9,9E9]],speeddata0,DefaultBlend,tool0;
  MoveAbsJ [[170.98,-54.91,-133.05,-21.79,-81.29,83.20],[9E9,9E9,9E9,9E9,9E9,9E9]],speeddata0,DefaultBlend,tool0;
  MoveAbsJ [[170.57,-54.63,-133.59,-22.78,-80.99,82.89],[9E9,9E9,9E9,9E9,9E9,9E9]],speeddata0,DefaultBlend,tool0;
  MoveAbsJ [[170.16,-54.34,-134.14,-23.77,-80.70,82.59],[9E9,9E9,9E9,9E9,9E9,9E9]],speeddata0,DefaultBlend,tool0;
  MoveAbsJ [[169.75,-54.06,-134.69,-24.76,-80.40,82.28],[9E9,9E9,9E9,9E9,9E9,9E9]],speeddata0,DefaultBlend,tool0;
  MoveAbsJ [[169.34,-53.77,-135.23,-25.75,-80.11,81.97],[9E9,9E9,9E9,9E9,9E9,9E9]],speeddata0,DefaultBlend,tool0;
  MoveAbsJ [[168.93,-53.49,-135.78,-26.74,-79.81,81.66],[9E9,9E9,9E9,9E9,9E9,9E9]],speeddata0,DefaultBlend,tool0;
  MoveAbsJ [[168.52,-53.21,-136.32,-27.73,-79.52,81.35],[9E9,9E9,9E9,9E9,9E9,9E9]],speeddata0,DefaultBlend,tool0;
  MoveAbsJ [[168.11,-52.92,-136.87,-28.72,-79.22,81.04],[9E9,9E9,9E9,9E9,9E9,9E9]],speeddata0,DefaultBlend,tool0;
  MoveAbsJ [[167.70,-52.64,-137.41,-29.71,-78.93,80.73],[9E9,9E9,9E9,9E9,9E9,9E9]],speeddata0,DefaultBlend,tool0;
  MoveAbsJ [[167.29,-52.35,-137.96,-30.70,-78.63,80.42],[9E9,9E9,9E9,9E9,9E9,9E9]],speeddata0,DefaultBlend,tool0;
  MoveAbsJ [[166.88,-52.07,-138.50,-31.69,-78.34,80.11],[9E9,9E9,9E9,9E9,9E9,9E9]],speeddata0,DefaultBlend,tool0;
  MoveAbsJ [[166.47,-51.78,-139.05,-32.68,-78.04,79.81],[9E9,9E9,9E9,9E9,9E9,9E9]],speeddata0,DefaultBlend,tool0;
  MoveAbsJ [[166.06,-51.50,-139.59,-33.67,-77.75,79.50],[9E9,9E9,9E9,9E9,9E9,9E9]],speeddata0,DefaultBlend,tool0;
  MoveAbsJ [[165.65,-51.21,-140.14,-34.66,-77.45,79.19],[9E9,9E9,9E9,9E9,9E9,9E9]],speeddata0,DefaultBlend,tool0;
  MoveAbsJ [[165.24,-50.93,-140.69,-35.65,-77.16,78.88],[9E9,9E9,9E9,9E9,9E9,9E9]],speeddata0,DefaultBlend,tool0;
  MoveAbsJ [[164.83,-50.64,-141.23,-36.64,-76.86,78.57],[9E9,9E9,9E9,9E9,9E9,9E9]],speeddata0,DefaultBlend,tool0;
  MoveAbsJ [[164.42,-50.36,-141.78,-37.63,-76.57,78.26],[9E9,9E9,9E9,9E9,9E9,9E9]],speeddata0,DefaultBlend,tool0;
  MoveAbsJ [[164.01,-50.07,-142.32,-38.62,-76.28,77.95],[9E9,9E9,9E9,9E9,9E9,9E9]],speeddata0,DefaultBlend,tool0;
  MoveAbsJ [[163.60,-49.79,-142.87,-39.61,-75.98,77.64],[9E9,9E9,9E9,9E9,9E9,9E9]],speeddata0,DefaultBlend,tool0;
  MoveAbsJ [[163.19,-49.51,-143.41,-40.60,-75.69,77.33],[9E9,9E9,9E9,9E9,9E9,9E9]],speeddata0,DefaultBlend,tool0;
  MoveAbsJ [[162.78,-49.22,-143.96,-41.59,-75.39,77.02],[9E9,9E9,9E9,9E9,9E9,9E9]],speeddata0,DefaultBlend,tool0;
  MoveAbsJ [[162.37,-48.94,-144.50,-42.58,-75.10,76.72],[9E9,9E9,9E9,9E9,9E9,9E9]],speeddata0,DefaultBlend,tool0;
  MoveAbsJ [[161.96,-48.65,-145.05,-43.57,-74.80,76.41],[9E9,9E9,9E9,9E9,9E9,9E9]],speeddata0,DefaultBlend,tool0;
  MoveAbsJ [[161.55,-48.37,-145.59,-44.56,-74.51,76.10],[9E9,9E9,9E9,9E9,9E9,9E9]],speeddata0,DefaultBlend,tool0;
  MoveAbsJ [[161.14,-48.08,-146.14,-45.55,-74.21,75.79],[9E9,9E9,9E9,9E9,9E9,9E9]],speeddata0,DefaultBlend,tool0;
  MoveAbsJ [[160.73,-47.80,-146.69,-46.54,-73.92,75.48],[9E9,9E9,9E9,9E9,9E9,9E9]],speeddata0,DefaultBlend,tool0;
  MoveAbsJ [[160.32,-47.51,-147.23,-47.53,-73.62,75.17],[9E9,9E9,9E9,9E9,9E9,9E9]],speeddata0,DefaultBlend,tool0;
  MoveAbsJ [[159.91,-47.23,-147.78,-48.52,-73.33,74.86],[9E9,9E9,9E9,9E9,9E9,9E9]],speeddata0,DefaultBlend,tool0;
  MoveAbsJ [[159.50,-46.94,-148.32,-49.51,-73.03,74.55],[9E9,9E9,9E9,9E9,9E9,9E9]],speeddata0,DefaultBlend,tool0;
  MoveAbsJ [[159.09,-46.66,-148.87,-50.50,-72.74,74.24],[9E9,9E9,9E9,9E9,9E9,9E9]],speeddata0,DefaultBlend,tool0;
  MoveAbsJ [[158.68,-46.38,-149.41,-51.49,-72.44,73.94],[9E9,9E9,9E9,9E9,9E9,9E9]],speeddata0,DefaultBlend,tool0;
  MoveAbsJ [[158.27,-46.09,-149.96,-52.48,-72.15,73.63],[9E9,9E9,9E9,9E9,9E9,9E9]],speeddata0,DefaultBlend,tool0;
  MoveAbsJ [[157.86,-45.81,-150.50,-53.47,-71.85,73.32],[9E9,9E9,9E9,9E9,9E9,9E9]],speeddata0,DefaultBlend,tool0;
  MoveAbsJ [[157.45,-45.52,-151.05,-54.46,-71.56,73.01],[9E9,9E9,9E9,9E9,9E9,9E9]],speeddata0,DefaultBlend,tool0;
  MoveAbsJ [[157.04,-45.24,-151.59,-55.45,-71.26,72.70],[9E9,9E9,9E9,9E9,9E9,9E9]],speeddata0,DefaultBlend,tool0;
  MoveAbsJ [[156.63,-44.95,-152.14,-56.44,-70.97,72.39],[9E9,9E9,9E9,9E9,9E9,9E9]],speeddata0,DefaultBlend,tool0;
  MoveAbsJ [[156.22,-44.67,-152.69,-57.43,-70.67,72.08],[9E9,9E9,9E9,9E9,9E9,9E9]],speeddata0,DefaultBlend,tool0;
  MoveAbsJ [[155.81,-44.38,-153.23,-58.42,-70.38,71.77],[9E9,9E9,9E9,9E9,9E9,9E9]],speeddata0,DefaultBlend,tool0;
  MoveAbsJ [[155.40,-44.10,-153.78,-59.42,-70.08,71.46],[9E9,9E9,9E9,9E9,9E9,9E9]],speeddata0,DefaultBlend,tool0;
  MoveAbsJ [[154.99,-43.81,-154.32,-60.41,-69.79,71.15],[9E9,9E9,9E9,9E9,9E9,9E9]],speeddata0,DefaultBlend,tool0;
  MoveAbsJ [[154.58,-43.53,-154.87,-61.40,-69.49,70.85],[9E9,9E9,9E9,9E9,9E9,9E9]],speeddata0,DefaultBlend,tool0;
  MoveAbsJ [[154.17,-43.25,-155.41,-62.39,-69.20,70.54],[9E9,9E9,9E9,9E9,9E9,9E9]],speeddata0,DefaultBlend,tool0;
  MoveAbsJ [[153.76,-42.96,-155.96,-63.38,-68.90,70.23],[9E9,9E9,9E9,9E9,9E9,9E9]],speeddata0,DefaultBlend,tool0;
  MoveAbsJ [[153.35,-42.68,-156.50,-64.37,-68.61,69.92],[9E9,9E9,9E9,9E9,9E9,9E9]],speeddata0,DefaultBlend,tool0;
  MoveAbsJ [[152.94,-42.39,-157.05,-65.36,-68.32,69.61],[9E9,9E9,9E9,9E9,9E9,9E9]],speeddata0,DefaultBlend,tool0;
  MoveAbsJ [[152.53,-42.11,-157.59,-66.35,-68.02,69.30],[9E9,9E9,9E9,9E9,9E9,9E9]],speeddata0,DefaultBlend,tool0;
  MoveAbsJ [[152.12,-41.82,-158.14,-67.34,-67.73,68.99],[9E9,9E9,9E9,9E9,9E9,9E9]],speeddata0,DefaultBlend,tool0;
  MoveAbsJ [[151.71,-41.54,-158.69,-68.33,-67.43,68.68],[9E9,9E9,9E9,9E9,9E9,9E9]],speeddata0,DefaultBlend,tool0;
  MoveAbsJ [[151.30,-41.25,-159.23,-69.32,-67.14,68.37],[9E9,9E9,9E9,9E9,9E9,9E9]],speeddata0,DefaultBlend,tool0;
  MoveAbsJ [[150.89,-40.97,-159.78,-70.31,-66.84,68.07],[9E9,9E9,9E9,9E9,9E9,9E9]],speeddata0,DefaultBlend,tool0;
  MoveAbsJ [[150.48,-40.68,-160.32,-71.30,-66.55,67.76],[9E9,9E9,9E9,9E9,9E9,9E9]],speeddata0,DefaultBlend,tool0;
  MoveAbsJ [[150.07,-40.40,-160.87,-72.29,-66.25,67.45],[9E9,9E9,9E9,9E9,9E9,9E9]],speeddata0,DefaultBlend,tool0;
  MoveAbsJ [[149.66,-40.12,-161.41,-73.28,-65.96,67.14],[9E9,9E9,9E9,9E9,9E9,9E9]],speeddata0,DefaultBlend,tool0;
  MoveAbsJ [[149.25,-39.83,-161.96,-74.27,-65.66,66.83],[9E9,9E9,9E9,9E9,9E9,9E9]],speeddata0,DefaultBlend,tool0;
  MoveAbsJ [[148.84,-39.55,-162.50,-75.26,-65.37,66.52],[9E9,9E9,9E9,9E9,9E9,9E9]],speeddata0,DefaultBlend,tool0;
  MoveAbsJ [[148.43,-39.26,-163.05,-76.25,-65.07,66.21],[9E9,9E9,9E9,9E9,9E9,9E9]],speeddata0,DefaultBlend,tool0;
  MoveAbsJ [[148.02,-38.98,-163.59,-77.24,-64.78,65.90],[9E9,9E9,9E9,9E9,9E9,9E9]],speeddata0,DefaultBlend,tool0;
  MoveAbsJ [[147.61,-38.69,-164.14,-78.23,-64.48,65.59],[9E9,9E9,9E9,9E9,9E9,9E9]],speeddata0,DefaultBlend,tool0;
  MoveAbsJ [[147.20,-38.41,-164.69,-79.22,-64.19,65.29],[9E9,9E9,9E9,9E9,9E9,9E9]],speeddata0,DefaultBlend,tool0;
  MoveAbsJ [[146.79,-38.12,-165.23,-80.21,-63.89,64.98],[9E9,9E9,9E9,9E9,9E9,9E9]],speeddata0,DefaultBlend,tool0;
  MoveAbsJ [[146.38,-37.84,-165.78,-81.20,-63.60,64.67],[9E9,9E9,9E9,9E9,9E9,9E9]],speeddata0,DefaultBlend,tool0;
  MoveAbsJ [[145.97,-37.55,-166.32,-82.19,-63.30,64.36],[9E9,9E9,9E9,9E9,9E9,9E9]],speeddata0,DefaultBlend,tool0;
  MoveAbsJ [[145.56,-37.27,-166.87,-83.18,-63.01,64.05],[9E9,9E9,9E9,9E9,9E9,9E9]],speeddata0,DefaultBlend,tool0;
  MoveAbsJ [[145.15,-36.99,-167.41,-84.17,-62.71,63.74],[9E9,9E9,9E9,9E9,9E9,9E9]],speeddata0,DefaultBlend,tool0;
  MoveAbsJ [[144.74,-36.70,-167.96,-85.16,-62.42,63.43],[9E9,9E9,9E9,9E9,9E9,9E9]],speeddata0,DefaultBlend,tool0;
  MoveAbsJ [[144.33,-36.42,-168.50,-86.15,-62.12,63.12],[9E9,9E9,9E9,9E9,9E9,9E9]],speeddata0,DefaultBlend,tool0;
  MoveAbsJ [[143.92,-36.13,-169.05,-87.14,-61.83,62.81],[9E9,9E9,9E9,9E9,9E9,9E9]],speeddata0,DefaultBlend,tool0;
  MoveAbsJ [[143.51,-35.85,-169.59,-88.13,-61.53,62.50],[9E9,9E9,9E9,9E9,9E9,9E9]],speeddata0,DefaultBlend,tool0;
  MoveAbsJ [[143.10,-35.56,-170.14,-89.12,-61.24,62.20],[9E9,9E9,9E9,9E9,9E9,9E9]],speeddata0,DefaultBlend,tool0;
  MoveAbsJ [[142.69,-35.28,-170.69,-90.11,-60.94,61.89],[9E9,9E9,9E9,9E9,9E9,9E9]],speeddata0,DefaultBlend,tool0;
  MoveAbsJ [[142.28,-34.99,-171.23,-91.10,-60.65,61.58],[9E9,9E9,9E9,9E9,9E9,9E9]],speeddata0,DefaultBlend,tool0;
  MoveAbsJ [[141.87,-34.71,-171.78,-92.09,-60.36,61.27],[9E9,9E9,9E9,9E9,9E9,9E9]],speeddata0,DefaultBlend,tool0;
  MoveAbsJ [[141.46,-34.42,-172.32,-93.08,-60.06,60.96],[9E9,9E9,9E9,9E9,9E9,9E9]],speeddata0,DefaultBlend,tool0;
  MoveAbsJ [[141.05,-34.14,-172.87,-94.07,-59.77,60.65],[9E9,9E9,9E9,9E9,9E9,9E9]],speeddata0,DefaultBlend,tool0;
  MoveAbsJ [[140.64,-33.86,-173.41,-95.06,-59.47,60.34],[9E9,9E9,9E9,9E9,9E9,9E9]],speeddata0,DefaultBlend,tool0;
  MoveAbsJ [[140.23,-33.57,-173.96,-96.05,-59.18,60.03],[9E9,9E9,9E9,9E9,9E9,9E9]],speeddata0,DefaultBlend,tool0;
  MoveAbsJ [[139.82,-33.29,-174.50,-97.04,-58.88,59.72],[9E9,9E9,9E9,9E9,9E9,9E9]],speeddata0,DefaultBlend,tool0;
  MoveAbsJ [[139.41,-33.00,-175.05,-98.03,-58.59,59.42],[9E9,9E9,9E9,9E9,9E9,9E9]],speeddata0,DefaultBlend,tool0;
  MoveAbsJ [[139.00,-32.72,-175.59,-99.03,-58.29,59.11],[9E9,9E9,9E9,9E9,9E9,9E9]],speeddata0,DefaultBlend,tool0;
  MoveAbsJ [[138.59,-32.43,-176.14,-100.02,-58.00,58.80],[9E9,9E9,9E9,9E9,9E9,9E9]],speeddata0,DefaultBlend,tool0;
  MoveAbsJ [[138.18,-32.15,-176.69,-101.01,-57.70,58.49],[9E9,9E9,9E9,9E9,9E9,9E9]],speeddata0,DefaultBlend,tool0;
  MoveAbsJ [[137.77,-31.86,-177.23,-102.00,-57.41,58.18],[9E9,9E9,9E9,9E9,9E9,9E9]],speeddata0,DefaultBlend,tool0;
  MoveAbsJ [[137.36,-31.58,-177.78,-102.99,-57.11,57.87],[9E9,9E9,9E9,9E9,9E9,9E9]],speeddata0,DefaultBlend,tool0;
  MoveAbsJ [[136.95,-31.29,-178.32,-103.98,-56.82,57.56],[9E9,9E9,9E9,9E9,9E9,9E9]],speeddata0,DefaultBlend,tool0;
  MoveAbsJ [[136.54,-31.01,-178.87,-104.97,-56.52,57.25],[9E9,9E9,9E9,9E9,9E9,9E9]],speeddata0,DefaultBlend,tool0;
  MoveAbsJ [[136.13,-30.72,-179.41,-105.96,-56.23,56.94],[9E9,9E9,9E9,9E9,9E9,9E9]],speeddata0,DefaultBlend,tool0;
  MoveAbsJ [[135.72,-30.44,-179.96,-106.95,-55.93,56.64],[9E9,9E9,9E9,9E9,9E9,9E9]],speeddata0,DefaultBlend,tool0;
  MoveAbsJ [[135.31,-30.16,-180.50,-107.94,-55.64,56.33],[9E9,9E9,9E9,9E9,9E9,9E9]],speeddata0,DefaultBlend,tool0;
  MoveAbsJ [[134.90,-29.87,-181.05,-108.93,-55.34,56.02],[9E9,9E9,9E9,9E9,9E9,9E9]],speeddata0,DefaultBlend,tool0;
  MoveAbsJ [[134.49,-29.59,-181.59,-109.92,-55.05,55.71],[9E9,9E9,9E9,9E9,9E9,9E9]],speeddata0,DefaultBlend,tool0;
  MoveAbsJ [[134.08,-29.30,-182.14,-110.91,-54.75,55.40],[9E9,9E9,9E9,9E9,9E9,9E9]],speeddata0,DefaultBlend,tool0;
  MoveAbsJ [[133.67,-29.02,-182.69,-111.90,-54.46,55.09],[9E9,9E9,9E9,9E9,9E9,9E9]],speeddata0,DefaultBlend,tool0;
  MoveAbsJ [[133.26,-28.73,-183.23,-112.89,-54.16,54.78],[9E9,9E9,9E9,9E9,9E9,9E9]],speeddata0,DefaultBlend,tool0;
  MoveAbsJ [[132.85,-28.45,-183.78,-113.88,-53.87,54.47],[9E9,9E9,9E9,9E9,9E9,9E9]],speeddata0,DefaultBlend,tool0;
  MoveAbsJ [[132.44,-28.16,-184.32,-114.87,-53.57,54.16],[9E9,9E9,9E9,9E9,9E9,9E9]],speeddata0,DefaultBlend,tool0;
  MoveAbsJ [[132.03,-27.88,-184.87,-115.86,-53.28,53.85],[9E9,9E9,9E9,9E9,9E9,9E9]],speeddata0,DefaultBlend,tool0;
  MoveAbsJ [[131.62,-27.59,-185.41,-116.85,-52.99,53.55],[9E9,9E9,9E9,9E9,9E9,9E9]],speeddata0,DefaultBlend,tool0;
  MoveAbsJ [[131.21,-27.31,-185.96,-117.84,-52.69,53.24],[9E9,9E9,9E9,9E9,9E9,9E9]],speeddata0,DefaultBlend,tool0;
  MoveAbsJ [[130.80,-27.03,-186.50,-118.83,-52.40,52.93],[9E9,9E9,9E9,9E9,9E9,9E9]],speeddata0,DefaultBlend,tool0;
  MoveAbsJ [[130.39,-26.74,-187.05,-119.82,-52.10,52.62],[9E9,9E9,9E9,9E9,9E9,9E9]],speeddata0,DefaultBlend,tool0;
  MoveAbsJ [[129.98,-26.46,-187.59,-120.81,-51.81,52.31],[9E9,9E9,9E9,9E9,9E9,9E9]],speeddata0,DefaultBlend,tool0;
  MoveAbsJ [[129.57,-26.17,-188.14,-121.80,-51.51,52.00],[9E9,9E9,9E9,9E9,9E9,9E9]],speeddata0,DefaultBlend,tool0;
  MoveAbsJ [[129.16,-25.89,-188.69,-122.79,-51.22,51.69],[9E9,9E9,9E9,9E9,9E9,9E9]],speeddata0,DefaultBlend,tool0;
  MoveAbsJ [[128.75,-25.60,-189.23,-123.78,-50.92,51.38],[9E9,9E9,9E9,9E9,9E9,9E9]],speeddata0,DefaultBlend,tool0;
  MoveAbsJ [[128.34,-25.32,-189.78,-124.77,-50.63,51.07],[9E9,9E9,9E9,9E9,9E9,9E9]],speeddata0,DefaultBlend,tool0;
  MoveAbsJ [[127.93,-25.03,-190.32,-125.76,-50.33,50.77],[9E9,9E9,9E9,9E9,9E9,9E9]],speeddata0,DefaultBlend,tool0;
  MoveAbsJ [[127.52,-24.75,-190.87,-126.75,-50.04,50.46],[9E9,9E9,9E9,9E9,9E9,9E9]],speeddata0,DefaultBlend,tool0;
  MoveAbsJ [[127.11,-24.46,-191.41,-127.74,-49.74,50.15],[9E9,9E9,9E9,9E9,9E9,9E9]],speeddata0,FinePoint,tool0;
  TPWrite "Action 29 LoadWorkpiece.";
  TPWrite "Press Play to Continue";
  Stop;
  TPWrite "Action 30 CloseGripper.";
  TPWrite "Press Play to Continue";
  Stop;
  TPWrite "Action 31 FreeMovement.";
  MoveAbsJ [[127.11,-24.46,-191.41,-127.74,-49.74,50.15],[9E9,9E9,9E9,9E9,9E9,9E9]],speeddata0,DefaultBlend,tool0;
  MoveAbsJ [[127.43,-24.63,-191.03,-126.75,-49.99,49.68],[9E9,9E9,9E9,9E9,9E9,9E9]],speeddata0,DefaultBlend,tool0;
  MoveAbsJ [[127.76,-24.79,-190.66,-125.76,-50.24,49.21],[9E9,9E9,9E9,9E9,9E9,9E9]],speeddata0,DefaultBlend,tool0;
  MoveAbsJ [[128.09,-24.95,-190.28,-124.77,-50.49,48.74],[9E9,9E9,9E9,9E9,9E9,9E9]],speeddata0,DefaultBlend,tool0;
  MoveAbsJ [[128.42,-25.12,-189.90,-123.78,-50.74,48.27],[9E9,9E9,9E9,9E9,9E9,9E9]],speeddata0,DefaultBlend,tool0;
  MoveAbsJ [[128.75,-25.28,-189.52,-122.79,-50.99,47.80],[9E9,9E9,9E9,9E9,9E9,9E9]],speeddata0,DefaultBlend,tool0;
  MoveAbsJ [[129.08,-25.44,-189.14,-121.80,-51.24,47.33],[9E9,9E9,9E9,9E9,9E9,9E9]],speeddata0,DefaultBlend,tool0;
  MoveAbsJ [[129.41,-25.61,-188.76,-120.81,-51.49,46.86],[9E9,9E9,9E9,9E9,9E9,9E9]],speeddata0,DefaultBlend,tool0;
  MoveAbsJ [[129.74,-25.77,-188.38,-119.82,-51.74,46.39],[9E9,9E9,9E9,9E9,9E9,9E9]],speeddata0,DefaultBlend,tool0;
  MoveAbsJ [[130.06,-25.93,-188.01,-118.83,-51.99,45.92],[9E9,9E9,9E9,9E9,9E9,9E9]],speeddata0,DefaultBlend,tool0;
  MoveAbsJ [[130.39,-26.10,-187.63,-117.84,-52.24,45.45],[9E9,9E9,9E9,9E9,9E9,9E9]],speeddata0,DefaultBlend,tool0;
  MoveAbsJ [[130.72,-26.26,-187.25,-116.85,-52.48,44.98],[9E9,9E9,9E9,9E9,9E9,9E9]],speeddata0,DefaultBlend,tool0;
  MoveAbsJ [[131.05,-26.42,-186.87,-115.86,-52.73,44.51],[9E9,9E9,9E9,9E9,9E9,9E9]],speeddata0,DefaultBlend,tool0;
  MoveAbsJ [[131.38,-26.59,-186.49,-114.87,-52.98,44.04],[9E9,9E9,9E9,9E9,9E9,9E9]],speeddata0,DefaultBlend,tool0;
  MoveAbsJ [[131.71,-26.75,-186.11,-113.88,-53.23,43.57],[9E9,9E9,9E9,9E9,9E9,9E9]],speeddata0,DefaultBlend,tool0;
  MoveAbsJ [[132.04,-26.91,-185.74,-112.89,-53.48,43.10],[9E9,9E9,9E9,9E9,9E9,9E9]],speeddata0,DefaultBlend,tool0;
  MoveAbsJ [[132.37,-27.08,-185.36,-111.90,-53.73,42.63],[9E9,9E9,9E9,9E9,9E9,9E9]],speeddata0,DefaultBlend,tool0;
  MoveAbsJ [[132.69,-27.24,-184.98,-110.91,-53.98,42.16],[9E9,9E9,9E9,9E9,9E9,9E9]],speeddata0,DefaultBlend,tool0;
  MoveAbsJ [[133.02,-27.40,-184.60,-109.92,-54.23,41.69],[9E9,9E9,9E9,9E9,9E9,9E9]],speeddata0,DefaultBlend,tool0;
  MoveAbsJ [[133.35,-27.56,-184.22,-108.93,-54.48,41.22],[9E9,9E9,9E9,9E9,9E9,9E9]],speeddata0,DefaultBlend,tool0;
  MoveAbsJ [[133.68,-27.73,-183.84,-107.94,-54.73,40.75],[9E9,9E9,9E9,9E9,9E9,9E9]],speeddata0,DefaultBlend,tool0;
  MoveAbsJ [[134.01,-27.89,-183.46,-106.95,-54.98,40.28],[9E9,9E9,9E9,9E9,9E9,9E9]],speeddata0,DefaultBlend,tool0;
  MoveAbsJ [[134.34,-28.05,-183.09,-105.96,-55.23,39.81],[9E9,9E9,9E9,9E9,9E9,9E9]],speeddata0,DefaultBlend,tool0;
  MoveAbsJ [[134.67,-28.22,-182.71,-104.97,-55.48,39.34],[9E9,9E9,9E9,9E9,9E9,9E9]],speeddata0,DefaultBlend,tool0;
  MoveAbsJ [[134.99,-28.38,-182.33,-103.98,-55.73,38.87],[9E9,9E9,9E9,9E9,9E9,9E9]],speeddata0,DefaultBlend,tool0;
  MoveAbsJ [[135.32,-28.54,-181.95,-102.99,-55.97,38.40],[9E9,9E9,9E9,9E9,9E9,9E9]],speeddata0,DefaultBlend,tool0;
  MoveAbsJ [[135.65,-28.71,-181.57,-102.00,-56.22,37.93],[9E9,9E9,9E9,9E9,9E9,9E9]],speeddata0,DefaultBlend,tool0;
  MoveAbsJ [[135.98,-28.87,-181.19,-101.01,-56.47,37.46],[9E9,9E9,9E9,9E9,9E9,9E9]],speeddata0,DefaultBlend,tool0;
  MoveAbsJ [[136.31,-29.03,-180.81,-100.02,-56.72,36.99],[9E9,9E9,9E9,9E9,9E9,9E9]],speeddata0,DefaultBlend,tool0;
  MoveAbsJ [[136.64,-29.20,-180.44,-99.03,-56.97,36.52],[9E9,9E9,9E9,9E9,9E9,9E9]],speeddata0,DefaultBlend,tool0;
  MoveAbsJ [[136.97,-29.36,-180.06,-98.03,-57.22,36.05],[9E9,9E9,9E9,9E9,9E9,9E9]],speeddata0,DefaultBlend,tool0;
  MoveAbsJ [[137.30,-29.52,-179.68,-97.04,-57.47,35.58],[9E9,9E9,9E9,9E9,9E9,9E9]],speeddata0,DefaultBlend,tool0;
  MoveAbsJ [[137.62,-29.69,-179.30,-96.05,-57.72,35.11],[9E9,9E9,9E9,9E9,9E9,9E9]],speeddata0,DefaultBlend,tool0;
  MoveAbsJ [[137.95,-29.85,-178.92,-95.06,-57.97,34.64],[9E9,9E9,9E9,9E9,9E9,9E9]],speeddata0,DefaultBlend,tool0;
  MoveAbsJ [[138.28,-30.01,-178.54,-94.07,-58.22,34.17],[9E9,9E9,9E9,9E9,9E9,9E9]],speeddata0,DefaultBlend,tool0;
  MoveAbsJ [[138.61,-30.18,-178.17,-93.08,-58.47,33.70],[9E9,9E9,9E9,9E9,9E9,9E9]],speeddata0,DefaultBlend,tool0;
  MoveAbsJ [[138.94,-30.34,-177.79,-92.09,-58.72,33.22],[9E9,9E9,9E9,9E9,9E9,9E9]],speeddata0,DefaultBlend,tool0;
  MoveAbsJ [[139.27,-30.50,-177.41,-91.10,-58.97,32.75],[9E9,9E9,9E9,9E9,9E9,9E9]],speeddata0,DefaultBlend,tool0;
  MoveAbsJ [[139.60,-30.66,-177.03,-90.11,-59.22,32.28],[9E9,9E9,9E9,9E9,9E9,9E9]],speeddata0,DefaultBlend,tool0;
  MoveAbsJ [[139.93,-30.83,-176.65,-89.12,-59.46,31.81],[9E9,9E9,9E9,9E9,9E9,9E9]],speeddata0,DefaultBlend,tool0;
  MoveAbsJ [[140.25,-30.99,-176.27,-88.13,-59.71,31.34],[9E9,9E9,9E9,9E9,9E9,9E9]],speeddata0,DefaultBlend,tool0;
  MoveAbsJ [[140.58,-31.15,-175.89,-87.14,-59.96,30.87],[9E9,9E9,9E9,9E9,9E9,9E9]],speeddata0,DefaultBlend,tool0;
  MoveAbsJ [[140.91,-31.32,-175.52,-86.15,-60.21,30.40],[9E9,9E9,9E9,9E9,9E9,9E9]],speeddata0,DefaultBlend,tool0;
  MoveAbsJ [[141.24,-31.48,-175.14,-85.16,-60.46,29.93],[9E9,9E9,9E9,9E9,9E9,9E9]],speeddata0,DefaultBlend,tool0;
  MoveAbsJ [[141.57,-31.64,-174.76,-84.17,-60.71,29.46],[9E9,9E9,9E9,9E9,9E9,9E9]],speeddata0,DefaultBlend,tool0;
  MoveAbsJ [[141.90,-31.81,-174.38,-83.18,-60.96,28.99],[9E9,9E9,9E9,9E9,9E9,9E9]],speeddata0,DefaultBlend,tool0;
  MoveAbsJ [[142.23,-31.97,-174.00,-82.19,-61.21,28.52],[9E9,9E9,9E9,9E9,9E9,9E9]],speeddata0,DefaultBlend,tool0;
  MoveAbsJ [[142.55,-32.13,-173.62,-81.20,-61.46,28.05],[9E9,9E9,9E9,9E9,9E9,9E9]],speeddata0,DefaultBlend,tool0;
  MoveAbsJ [[142.88,-32.30,-173.25,-80.21,-61.71,27.58],[9E9,9E9,9E9,9E9,9E9,9E9]],speeddata0,DefaultBlend,tool0;
  MoveAbsJ [[143.21,-32.46,-172.87,-79.22,-61.96,27.11],[9E9,9E9,9E9,9E9,9E9,9E9]],speeddata0,DefaultBlend,tool0;
  MoveAbsJ [[143.54,-32.62,-172.49,-78.23,-62.21,26.64],[9E9,9E9,9E9,9E9,9E9,9E9]],speeddata0,DefaultBlend,tool0;
  MoveAbsJ [[143.87,-32.79,-172.11,-77.24,-62.46,26.17],[9E9,9E9,9E9,9E9,9E9,9E9]],speeddata0,DefaultBlend,tool0;
  MoveAbsJ [[144.20,-32.95,-171.73,-76.25,-62.71,25.70],[9E9,9E9,9E9,9E9,9E9,9E9]],speeddata0,DefaultBlend,tool0;
  MoveAbsJ [[144.53,-33.11,-171.35,-75.26,-62.95,25.23],[9E9,9E9,9E9,9E9,9E9,9E9]],speeddata0,DefaultBlend,tool0;
  MoveAbsJ [[144.86,-33.28,-170.97,-74.27,-63.20,24.76],[9E9,9E9,9E9,9E9,9E9,9E9]],speeddata0,DefaultBlend,tool0;
  MoveAbsJ [[145.18,-33.44,-170.60,-73.28,-63.45,24.29],[9E9,9E9,9E9,9E9,9E9,9E9]],speeddata0,DefaultBlend,tool0;
  MoveAbsJ [[145.51,-33.60,-170.22,-72.29,-63.70,23.82],[9E9,9E9,9E9,9E9,9E9,9E9]],speeddata0,DefaultBlend,tool0;
  MoveAbsJ [[145.84,-33.76,-169.84,-71.30,-63.95,23.35],[9E9,9E9,9E9,9E9,9E9,9E9]],speeddata0,DefaultBlend,tool0;
  MoveAbsJ [[146.17,-33.93,-169.46,-70.31,-64.20,22.88],[9E9,9E9,9E9,9E9,9E9,9E9]],speeddata0,DefaultBlend,tool0;
  MoveAbsJ [[146.50,-34.09,-169.08,-69.32,-64.45,22.41],[9E9,9E9,9E9,9E9,9E9,9E9]],speeddata0,DefaultBlend,tool0;
  MoveAbsJ [[146.83,-34.25,-168.70,-68.33,-64.70,21.94],[9E9,9E9,9E9,9E9,9E9,9E9]],speeddata0,DefaultBlend,tool0;
  MoveAbsJ [[147.16,-34.42,-168.32,-67.34,-64.95,21.47],[9E9,9E9,9E9,9E9,9E9,9E9]],speeddata0,DefaultBlend,tool0;
  MoveAbsJ [[147.49,-34.58,-167.95,-66.35,-65.20,21.00],[9E9,9E9,9E9,9E9,9E9,9E9]],speeddata0,DefaultBlend,tool0;
  MoveAbsJ [[147.81,-34.74,-167.57,-65.36,-65.45,20.53],[9E9,9E9,9E9,9E9,9E9,9E9]],speeddata0,DefaultBlend,tool0;
  MoveAbsJ [[148.14,-34.91,-167.19,-64.37,-65.70,20.06],[9E9,9E9,9E9,9E9,9E9,9E9]],speeddata0,DefaultBlend,tool0;
  MoveAbsJ [[148.47,-35.07,-166.81,-63.38,-65.95,19.59],[9E9,9E9,9E9,9E9,9E9,9E9]],speeddata0,DefaultBlend,tool0;
  MoveAbsJ [[148.80,-35.23,-166.43,-62.39,-66.20,19.12],[9E9,9E9,9E9,9E9,9E9,9E9]],speeddata0,DefaultBlend,tool0;
  MoveAbsJ [[149.13,-35.40,-166.05,-61.40,-66.44,18.65],[9E9,9E9,9E9,9E9,9E9,9E9]],speeddata0,DefaultBlend,tool0;
  MoveAbsJ [[149.46,-35.56,-165.68,-60.41,-66.69,18.18],[9E9,9E9,9E9,9E9,9E9,9E9]],speeddata0,DefaultBlend,tool0;
  MoveAbsJ [[149.79,-35.72,-165.30,-59.42,-66.94,17.71],[9E9,9E9,9E9,9E9,9E9,9E9]],speeddata0,DefaultBlend,tool0;
  MoveAbsJ [[150.12,-35.89,-164.92,-58.42,-67.19,17.24],[9E9,9E9,9E9,9E9,9E9,9E9]],speeddata0,DefaultBlend,tool0;
  MoveAbsJ [[150.44,-36.05,-164.54,-57.43,-67.44,16.77],[9E9,9E9,9E9,9E9,9E9,9E9]],speeddata0,DefaultBlend,tool0;
  MoveAbsJ [[150.77,-36.21,-164.16,-56.44,-67.69,16.30],[9E9,9E9,9E9,9E9,9E9,9E9]],speeddata0,DefaultBlend,tool0;
  MoveAbsJ [[151.10,-36.38,-163.78,-55.45,-67.94,15.83],[9E9,9E9,9E9,9E9,9E9,9E9]],speeddata0,DefaultBlend,tool0;
  MoveAbsJ [[151.43,-36.54,-163.40,-54.46,-68.19,15.36],[9E9,9E9,9E9,9E9,9E9,9E9]],speeddata0,DefaultBlend,tool0;
  MoveAbsJ [[151.76,-36.70,-163.03,-53.47,-68.44,14.89],[9E9,9E9,9E9,9E9,9E9,9E9]],speeddata0,DefaultBlend,tool0;
  MoveAbsJ [[152.09,-36.86,-162.65,-52.48,-68.69,14.42],[9E9,9E9,9E9,9E9,9E9,9E9]],speeddata0,DefaultBlend,tool0;
  MoveAbsJ [[152.42,-37.03,-162.27,-51.49,-68.94,13.95],[9E9,9E9,9E9,9E9,9E9,9E9]],speeddata0,DefaultBlend,tool0;
  MoveAbsJ [[152.74,-37.19,-161.89,-50.50,-69.19,13.48],[9E9,9E9,9E9,9E9,9E9,9E9]],speeddata0,DefaultBlend,tool0;
  MoveAbsJ [[153.07,-37.35,-161.51,-49.51,-69.44,13.01],[9E9,9E9,9E9,9E9,9E9,9E9]],speeddata0,DefaultBlend,tool0;
  MoveAbsJ [[153.40,-37.52,-161.13,-48.52,-69.69,12.54],[9E9,9E9,9E9,9E9,9E9,9E9]],speeddata0,DefaultBlend,tool0;
  MoveAbsJ [[153.73,-37.68,-160.75,-47.53,-69.94,12.07],[9E9,9E9,9E9,9E9,9E9,9E9]],speeddata0,DefaultBlend,tool0;
  MoveAbsJ [[154.06,-37.84,-160.38,-46.54,-70.18,11.60],[9E9,9E9,9E9,9E9,9E9,9E9]],speeddata0,DefaultBlend,tool0;
  MoveAbsJ [[154.39,-38.01,-160.00,-45.55,-70.43,11.13],[9E9,9E9,9E9,9E9,9E9,9E9]],speeddata0,DefaultBlend,tool0;
  MoveAbsJ [[154.72,-38.17,-159.62,-44.56,-70.68,10.66],[9E9,9E9,9E9,9E9,9E9,9E9]],speeddata0,DefaultBlend,tool0;
  MoveAbsJ [[155.05,-38.33,-159.24,-43.57,-70.93,10.19],[9E9,9E9,9E9,9E9,9E9,9E9]],speeddata0,DefaultBlend,tool0;
  MoveAbsJ [[155.37,-38.50,-158.86,-42.58,-71.18,9.72],[9E9,9E9,9E9,9E9,9E9,9E9]],speeddata0,DefaultBlend,tool0;
  MoveAbsJ [[155.70,-38.66,-158.48,-41.59,-71.43,9.25],[9E9,9E9,9E9,9E9,9E9,9E9]],speeddata0,DefaultBlend,tool0;
  MoveAbsJ [[156.03,-38.82,-158.11,-40.60,-71.68,8.78],[9E9,9E9,9E9,9E9,9E9,9E9]],speeddata0,DefaultBlend,tool0;
  MoveAbsJ [[156.36,-38.99,-157.73,-39.61,-71.93,8.31],[9E9,9E9,9E9,9E9,9E9,9E9]],speeddata0,DefaultBlend,tool0;
  MoveAbsJ [[156.69,-39.15,-157.35,-38.62,-72.18,7.84],[9E9,9E9,9E9,9E9,9E9,9E9]],speeddata0,DefaultBlend,tool0;
  MoveAbsJ [[157.02,-39.31,-156.97,-37.63,-72.43,7.37],[9E9,9E9,9E9,9E9,9E9,9E9]],speeddata0,DefaultBlend,tool0;
  MoveAbsJ [[157.35,-39.48,-156.59,-36.64,-72.68,6.90],[9E9,9E9,9E9,9E9,9E9,9E9]],speeddata0,DefaultBlend,tool0;
  MoveAbsJ [[157.68,-39.64,-156.21,-35.65,-72.93,6.43],[9E9,9E9,9E9,9E9,9E9,9E9]],speeddata0,DefaultBlend,tool0;
  MoveAbsJ [[158.00,-39.80,-155.83,-34.66,-73.18,5.96],[9E9,9E9,9E9,9E9,9E9,9E9]],speeddata0,DefaultBlend,tool0;
  MoveAbsJ [[158.33,-39.96,-155.46,-33.67,-73.43,5.49],[9E9,9E9,9E9,9E9,9E9,9E9]],speeddata0,DefaultBlend,tool0;
  MoveAbsJ [[158.66,-40.13,-155.08,-32.68,-73.67,5.02],[9E9,9E9,9E9,9E9,9E9,9E9]],speeddata0,DefaultBlend,tool0;
  MoveAbsJ [[158.99,-40.29,-154.70,-31.69,-73.92,4.55],[9E9,9E9,9E9,9E9,9E9,9E9]],speeddata0,DefaultBlend,tool0;
  MoveAbsJ [[159.32,-40.45,-154.32,-30.70,-74.17,4.08],[9E9,9E9,9E9,9E9,9E9,9E9]],speeddata0,DefaultBlend,tool0;
  MoveAbsJ [[159.65,-40.62,-153.94,-29.71,-74.42,3.61],[9E9,9E9,9E9,9E9,9E9,9E9]],speeddata0,DefaultBlend,tool0;
  MoveAbsJ [[159.98,-40.78,-153.56,-28.72,-74.67,3.14],[9E9,9E9,9E9,9E9,9E9,9E9]],speeddata0,DefaultBlend,tool0;
  MoveAbsJ [[160.30,-40.94,-153.19,-27.73,-74.92,2.67],[9E9,9E9,9E9,9E9,9E9,9E9]],speeddata0,DefaultBlend,tool0;
  MoveAbsJ [[160.63,-41.11,-152.81,-26.74,-75.17,2.20],[9E9,9E9,9E9,9E9,9E9,9E9]],speeddata0,DefaultBlend,tool0;
  MoveAbsJ [[160.96,-41.27,-152.43,-25.75,-75.42,1.73],[9E9,9E9,9E9,9E9,9E9,9E9]],speeddata0,DefaultBlend,tool0;
  MoveAbsJ [[161.29,-41.43,-152.05,-24.76,-75.67,1.26],[9E9,9E9,9E9,9E9,9E9,9E9]],speeddata0,DefaultBlend,tool0;
  MoveAbsJ [[161.62,-41.60,-151.67,-23.77,-75.92,0.79],[9E9,9E9,9E9,9E9,9E9,9E9]],speeddata0,DefaultBlend,tool0;
  MoveAbsJ [[161.95,-41.76,-151.29,-22.78,-76.17,0.32],[9E9,9E9,9E9,9E9,9E9,9E9]],speeddata0,DefaultBlend,tool0;
  MoveAbsJ [[162.28,-41.92,-150.91,-21.79,-76.42,-0.15],[9E9,9E9,9E9,9E9,9E9,9E9]],speeddata0,DefaultBlend,tool0;
  MoveAbsJ [[162.61,-42.09,-150.54,-20.80,-76.67,-0.62],[9E9,9E9,9E9,9E9,9E9,9E9]],speeddata0,DefaultBlend,tool0;
  MoveAbsJ [[162.93,-42.25,-150.16,-19.81,-76.92,-1.09],[9E9,9E9,9E9,9E9,9E9,9E9]],speeddata0,DefaultBlend,tool0;
  MoveAbsJ [[163.26,-42.41,-149.78,-18.81,-77.16,-1.56],[9E9,9E9,9E9,9E9,9E9,9E9]],speeddata0,DefaultBlend,tool0;
  MoveAbsJ [[163.59,-42.58,-149.40,-17.82,-77.41,-2.03],[9E9,9E9,9E9,9E9,9E9,9E9]],speeddata0,DefaultBlend,tool0;
  MoveAbsJ [[163.92,-42.74,-149.02,-16.83,-77.66,-2.50],[9E9,9E9,9E9,9E9,9E9,9E9]],speeddata0,DefaultBlend,tool0;
  MoveAbsJ [[164.25,-42.90,-148.64,-15.84,-77.91,-2.97],[9E9,9E9,9E9,9E9,9E9,9E9]],speeddata0,DefaultBlend,tool0;
  MoveAbsJ [[164.58,-43.06,-148.26,-14.85,-78.16,-3.44],[9E9,9E9,9E9,9E9,9E9,9E9]],speeddata0,DefaultBlend,tool0;
  MoveAbsJ [[164.91,-43.23,-147.89,-13.86,-78.41,-3.91],[9E9,9E9,9E9,9E9,9E9,9E9]],speeddata0,DefaultBlend,tool0;
  MoveAbsJ [[165.24,-43.39,-147.51,-12.87,-78.66,-4.38],[9E9,9E9,9E9,9E9,9E9,9E9]],speeddata0,DefaultBlend,tool0;
  MoveAbsJ [[165.56,-43.55,-147.13,-11.88,-78.91,-4.85],[9E9,9E9,9E9,9E9,9E9,9E9]],speeddata0,DefaultBlend,tool0;
  MoveAbsJ [[165.89,-43.72,-146.75,-10.89,-79.16,-5.32],[9E9,9E9,9E9,9E9,9E9,9E9]],speeddata0,DefaultBlend,tool0;
  MoveAbsJ [[166.22,-43.88,-146.37,-9.90,-79.41,-5.79],[9E9,9E9,9E9,9E9,9E9,9E9]],speeddata0,DefaultBlend,tool0;
  MoveAbsJ [[166.55,-44.04,-145.99,-8.91,-79.66,-6.26],[9E9,9E9,9E9,9E9,9E9,9E9]],speeddata0,DefaultBlend,tool0;
  MoveAbsJ [[166.88,-44.21,-145.62,-7.92,-79.91,-6.73],[9E9,9E9,9E9,9E9,9E9,9E9]],speeddata0,DefaultBlend,tool0;
  MoveAbsJ [[167.21,-44.37,-145.24,-6.93,-80.16,-7.20],[9E9,9E9,9E9,9E9,9E9,9E9]],speeddata0,DefaultBlend,tool0;
  MoveAbsJ [[167.54,-44.53,-144.86,-5.94,-80.41,-7.67],[9E9,9E9,9E9,9E9,9E9,9E9]],speeddata0,DefaultBlend,tool0;
  MoveAbsJ [[167.87,-44.70,-144.48,-4.95,-80.65,-8.14],[9E9,9E9,9E9,9E9,9E9,9E9]],speeddata0,DefaultBlend,tool0;
  MoveAbsJ [[168.19,-44.86,-144.10,-3.96,-80.90,-8.61],[9E9,9E9,9E9,9E9,9E9,9E9]],speeddata0,DefaultBlend,tool0;
  MoveAbsJ [[168.52,-45.02,-143.72,-2.97,-81.15,-9.08],[9E9,9E9,9E9,9E9,9E9,9E9]],speeddata0,DefaultBlend,tool0;
  MoveAbsJ [[168.85,-45.19,-143.34,-1.98,-81.40,-9.55],[9E9,9E9,9E9,9E9,9E9,9E9]],speeddata0,DefaultBlend,tool0;
  MoveAbsJ [[169.18,-45.35,-142.97,-0.99,-81.65,-10.02],[9E9,9E9,9E9,9E9,9E9,9E9]],speeddata0,DefaultBlend,tool0;
  MoveAbsJ [[169.51,-45.51,-142.59,-0.00,-81.90,-10.49],[9E9,9E9,9E9,9E9,9E9,9E9]],speeddata0,FinePoint,tool0;
  TPWrite "Action 32 LinearMovement.";
  MoveAbsJ [[169.51,-45.51,-142.59,-0.00,-81.90,-10.49],[9E9,9E9,9E9,9E9,9E9,9E9]],speeddata0,DefaultBlend,tool0;
  MoveAbsJ [[169.51,-46.03,-142.89,-0.00,-81.08,-10.49],[9E9,9E9,9E9,9E9,9E9,9E9]],speeddata0,DefaultBlend,tool0;
  MoveAbsJ [[169.51,-46.54,-143.22,-0.00,-80.24,-10.49],[9E9,9E9,9E9,9E9,9E9,9E9]],speeddata0,DefaultBlend,tool0;
  MoveAbsJ [[169.51,-47.06,-143.54,-0.00,-79.41,-10.49],[9E9,9E9,9E9,9E9,9E9,9E9]],speeddata0,DefaultBlend,tool0;
  MoveAbsJ [[169.51,-47.60,-143.82,-0.00,-78.58,-10.49],[9E9,9E9,9E9,9E9,9E9,9E9]],speeddata0,DefaultBlend,tool0;
  MoveAbsJ [[169.51,-48.15,-144.09,-0.00,-77.77,-10.49],[9E9,9E9,9E9,9E9,9E9,9E9]],speeddata0,DefaultBlend,tool0;
  MoveAbsJ [[169.51,-48.72,-144.32,-0.00,-76.97,-10.49],[9E9,9E9,9E9,9E9,9E9,9E9]],speeddata0,DefaultBlend,tool0;
  MoveAbsJ [[169.51,-49.30,-144.53,-0.00,-76.17,-10.49],[9E9,9E9,9E9,9E9,9E9,9E9]],speeddata0,DefaultBlend,tool0;
  MoveAbsJ [[169.51,-49.90,-144.72,-0.00,-75.39,-10.49],[9E9,9E9,9E9,9E9,9E9,9E9]],speeddata0,FinePoint,tool0;
  TPWrite "Action 33 OpenGripper.";
  TPWrite "Press Play to Continue";
  Stop;
  TPWrite "Action 34 LinearMovement.";
  MoveAbsJ [[169.51,-49.89,-144.73,-0.00,-75.38,-10.49],[9E9,9E9,9E9,9E9,9E9,9E9]],speeddata0,DefaultBlend,tool0;
  MoveAbsJ [[169.51,-49.26,-144.61,-0.00,-76.14,-10.49],[9E9,9E9,9E9,9E9,9E9,9E9]],speeddata0,DefaultBlend,tool0;
  MoveAbsJ [[169.51,-48.66,-144.42,-0.00,-76.92,-10.49],[9E9,9E9,9E9,9E9,9E9,9E9]],speeddata0,DefaultBlend,tool0;
  MoveAbsJ [[169.51,-48.09,-144.19,-0.00,-77.71,-10.49],[9E9,9E9,9E9,9E9,9E9,9E9]],speeddata0,DefaultBlend,tool0;
  MoveAbsJ [[169.51,-47.53,-143.95,-0.00,-78.52,-10.49],[9E9,9E9,9E9,9E9,9E9,9E9]],speeddata0,DefaultBlend,tool0;
  MoveAbsJ [[169.51,-46.99,-143.67,-0.00,-79.34,-10.49],[9E9,9E9,9E9,9E9,9E9,9E9]],speeddata0,DefaultBlend,tool0;
  MoveAbsJ [[169.51,-46.46,-143.37,-0.00,-80.16,-10.49],[9E9,9E9,9E9,9E9,9E9,9E9]],speeddata0,DefaultBlend,tool0;
  MoveAbsJ [[169.51,-45.95,-143.05,-0.00,-81.00,-10.49],[9E9,9E9,9E9,9E9,9E9,9E9]],speeddata0,DefaultBlend,tool0;
  MoveAbsJ [[169.51,-45.45,-142.69,-0.00,-81.85,-10.49],[9E9,9E9,9E9,9E9,9E9,9E9]],speeddata0,FinePoint,tool0;
  TPWrite "Action 35 FreeMovement.";
  MoveAbsJ [[169.51,-45.45,-142.69,-0.00,-81.85,-10.49],[9E9,9E9,9E9,9E9,9E9,9E9]],speeddata0,DefaultBlend,tool0;
  MoveAbsJ [[169.18,-45.29,-143.07,-0.99,-81.60,-10.02],[9E9,9E9,9E9,9E9,9E9,9E9]],speeddata0,DefaultBlend,tool0;
  MoveAbsJ [[168.85,-45.13,-143.45,-1.98,-81.35,-9.55],[9E9,9E9,9E9,9E9,9E9,9E9]],speeddata0,DefaultBlend,tool0;
  MoveAbsJ [[168.52,-44.97,-143.83,-2.97,-81.10,-9.08],[9E9,9E9,9E9,9E9,9E9,9E9]],speeddata0,DefaultBlend,tool0;
  MoveAbsJ [[168.19,-44.80,-144.21,-3.96,-80.85,-8.61],[9E9,9E9,9E9,9E9,9E9,9E9]],speeddata0,DefaultBlend,tool0;
  MoveAbsJ [[167.87,-44.64,-144.58,-4.95,-80.60,-8.14],[9E9,9E9,9E9,9E9,9E9,9E9]],speeddata0,DefaultBlend,tool0;
  MoveAbsJ [[167.54,-44.48,-144.96,-5.94,-80.35,-7.67],[9E9,9E9,9E9,9E9,9E9,9E9]],speeddata0,DefaultBlend,tool0;
  MoveAbsJ [[167.21,-44.32,-145.34,-6.93,-80.10,-7.20],[9E9,9E9,9E9,9E9,9E9,9E9]],speeddata0,DefaultBlend,tool0;
  MoveAbsJ [[166.88,-44.15,-145.72,-7.92,-79.86,-6.73],[9E9,9E9,9E9,9E9,9E9,9E9]],speeddata0,DefaultBlend,tool0;
  MoveAbsJ [[166.55,-43.99,-146.09,-8.91,-79.61,-6.26],[9E9,9E9,9E9,9E9,9E9,9E9]],speeddata0,DefaultBlend,tool0;
  MoveAbsJ [[166.22,-43.83,-146.47,-9.90,-79.36,-5.79],[9E9,9E9,9E9,9E9,9E9,9E9]],speeddata0,DefaultBlend,tool0;
  MoveAbsJ [[165.89,-43.66,-146.85,-10.89,-79.11,-5.32],[9E9,9E9,9E9,9E9,9E9,9E9]],speeddata0,DefaultBlend,tool0;
  MoveAbsJ [[165.56,-43.50,-147.23,-11.88,-78.86,-4.85],[9E9,9E9,9E9,9E9,9E9,9E9]],speeddata0,DefaultBlend,tool0;
  MoveAbsJ [[165.24,-43.34,-147.60,-12.87,-78.61,-4.38],[9E9,9E9,9E9,9E9,9E9,9E9]],speeddata0,DefaultBlend,tool0;
  MoveAbsJ [[164.91,-43.18,-147.98,-13.86,-78.36,-3.91],[9E9,9E9,9E9,9E9,9E9,9E9]],speeddata0,DefaultBlend,tool0;
  MoveAbsJ [[164.58,-43.01,-148.36,-14.85,-78.11,-3.44],[9E9,9E9,9E9,9E9,9E9,9E9]],speeddata0,DefaultBlend,tool0;
  MoveAbsJ [[164.25,-42.85,-148.74,-15.84,-77.86,-2.97],[9E9,9E9,9E9,9E9,9E9,9E9]],speeddata0,DefaultBlend,tool0;
  MoveAbsJ [[163.92,-42.69,-149.11,-16.83,-77.62,-2.50],[9E9,9E9,9E9,9E9,9E9,9E9]],speeddata0,DefaultBlend,tool0;
  MoveAbsJ [[163.59,-42.53,-149.49,-17.82,-77.37,-2.03],[9E9,9E9,9E9,9E9,9E9,9E9]],speeddata0,DefaultBlend,tool0;
  MoveAbsJ [[163.26,-42.36,-149.87,-18.81,-77.12,-1.56],[9E9,9E9,9E9,9E9,9E9,9E9]],speeddata0,DefaultBlend,tool0;
  MoveAbsJ [[162.93,-42.20,-150.25,-19.80,-76.87,-1.09],[9E9,9E9,9E9,9E9,9E9,9E9]],speeddata0,DefaultBlend,tool0;
  MoveAbsJ [[162.61,-42.04,-150.63,-20.79,-76.62,-0.62],[9E9,9E9,9E9,9E9,9E9,9E9]],speeddata0,DefaultBlend,tool0;
  MoveAbsJ [[162.28,-41.87,-151.00,-21.78,-76.37,-0.15],[9E9,9E9,9E9,9E9,9E9,9E9]],speeddata0,DefaultBlend,tool0;
  MoveAbsJ [[161.95,-41.71,-151.38,-22.77,-76.12,0.32],[9E9,9E9,9E9,9E9,9E9,9E9]],speeddata0,DefaultBlend,tool0;
  MoveAbsJ [[161.62,-41.55,-151.76,-23.77,-75.87,0.79],[9E9,9E9,9E9,9E9,9E9,9E9]],speeddata0,DefaultBlend,tool0;
  MoveAbsJ [[161.29,-41.39,-152.14,-24.76,-75.63,1.26],[9E9,9E9,9E9,9E9,9E9,9E9]],speeddata0,DefaultBlend,tool0;
  MoveAbsJ [[160.96,-41.22,-152.51,-25.75,-75.38,1.73],[9E9,9E9,9E9,9E9,9E9,9E9]],speeddata0,DefaultBlend,tool0;
  MoveAbsJ [[160.63,-41.06,-152.89,-26.74,-75.13,2.20],[9E9,9E9,9E9,9E9,9E9,9E9]],speeddata0,DefaultBlend,tool0;
  MoveAbsJ [[160.31,-40.90,-153.27,-27.73,-74.88,2.67],[9E9,9E9,9E9,9E9,9E9,9E9]],speeddata0,DefaultBlend,tool0;
  MoveAbsJ [[159.98,-40.74,-153.65,-28.72,-74.63,3.14],[9E9,9E9,9E9,9E9,9E9,9E9]],speeddata0,DefaultBlend,tool0;
  MoveAbsJ [[159.65,-40.57,-154.02,-29.71,-74.38,3.61],[9E9,9E9,9E9,9E9,9E9,9E9]],speeddata0,DefaultBlend,tool0;
  MoveAbsJ [[159.32,-40.41,-154.40,-30.70,-74.13,4.08],[9E9,9E9,9E9,9E9,9E9,9E9]],speeddata0,DefaultBlend,tool0;
  MoveAbsJ [[158.99,-40.25,-154.78,-31.69,-73.88,4.55],[9E9,9E9,9E9,9E9,9E9,9E9]],speeddata0,DefaultBlend,tool0;
  MoveAbsJ [[158.66,-40.08,-155.16,-32.68,-73.63,5.02],[9E9,9E9,9E9,9E9,9E9,9E9]],speeddata0,DefaultBlend,tool0;
  MoveAbsJ [[158.33,-39.92,-155.53,-33.67,-73.39,5.49],[9E9,9E9,9E9,9E9,9E9,9E9]],speeddata0,DefaultBlend,tool0;
  MoveAbsJ [[158.00,-39.76,-155.91,-34.66,-73.14,5.96],[9E9,9E9,9E9,9E9,9E9,9E9]],speeddata0,DefaultBlend,tool0;
  MoveAbsJ [[157.68,-39.60,-156.29,-35.65,-72.89,6.43],[9E9,9E9,9E9,9E9,9E9,9E9]],speeddata0,DefaultBlend,tool0;
  MoveAbsJ [[157.35,-39.43,-156.67,-36.64,-72.64,6.90],[9E9,9E9,9E9,9E9,9E9,9E9]],speeddata0,DefaultBlend,tool0;
  MoveAbsJ [[157.02,-39.27,-157.05,-37.63,-72.39,7.37],[9E9,9E9,9E9,9E9,9E9,9E9]],speeddata0,DefaultBlend,tool0;
  MoveAbsJ [[156.69,-39.11,-157.42,-38.62,-72.14,7.84],[9E9,9E9,9E9,9E9,9E9,9E9]],speeddata0,DefaultBlend,tool0;
  MoveAbsJ [[156.36,-38.95,-157.80,-39.61,-71.89,8.31],[9E9,9E9,9E9,9E9,9E9,9E9]],speeddata0,DefaultBlend,tool0;
  MoveAbsJ [[156.03,-38.78,-158.18,-40.60,-71.64,8.78],[9E9,9E9,9E9,9E9,9E9,9E9]],speeddata0,DefaultBlend,tool0;
  MoveAbsJ [[155.70,-38.62,-158.56,-41.59,-71.39,9.25],[9E9,9E9,9E9,9E9,9E9,9E9]],speeddata0,DefaultBlend,tool0;
  MoveAbsJ [[155.37,-38.46,-158.93,-42.58,-71.15,9.72],[9E9,9E9,9E9,9E9,9E9,9E9]],speeddata0,DefaultBlend,tool0;
  MoveAbsJ [[155.05,-38.29,-159.31,-43.57,-70.90,10.19],[9E9,9E9,9E9,9E9,9E9,9E9]],speeddata0,DefaultBlend,tool0;
  MoveAbsJ [[154.72,-38.13,-159.69,-44.56,-70.65,10.66],[9E9,9E9,9E9,9E9,9E9,9E9]],speeddata0,DefaultBlend,tool0;
  MoveAbsJ [[154.39,-37.97,-160.07,-45.55,-70.40,11.13],[9E9,9E9,9E9,9E9,9E9,9E9]],speeddata0,DefaultBlend,tool0;
  MoveAbsJ [[154.06,-37.81,-160.44,-46.54,-70.15,11.60],[9E9,9E9,9E9,9E9,9E9,9E9]],speeddata0,DefaultBlend,tool0;
  MoveAbsJ [[153.73,-37.64,-160.82,-47.53,-69.90,12.07],[9E9,9E9,9E9,9E9,9E9,9E9]],speeddata0,DefaultBlend,tool0;
  MoveAbsJ [[153.40,-37.48,-161.20,-48.52,-69.65,12.54],[9E9,9E9,9E9,9E9,9E9,9E9]],speeddata0,DefaultBlend,tool0;
  MoveAbsJ [[153.07,-37.32,-161.58,-49.51,-69.40,13.01],[9E9,9E9,9E9,9E9,9E9,9E9]],speeddata0,DefaultBlend,tool0;
  MoveAbsJ [[152.75,-37.16,-161.95,-50.50,-69.15,13.48],[9E9,9E9,9E9,9E9,9E9,9E9]],speeddata0,DefaultBlend,tool0;
  MoveAbsJ [[152.42,-36.99,-162.33,-51.49,-68.91,13.95],[9E9,9E9,9E9,9E9,9E9,9E9]],speeddata0,DefaultBlend,tool0;
  MoveAbsJ [[152.09,-36.83,-162.71,-52.48,-68.66,14.42],[9E9,9E9,9E9,9E9,9E9,9E9]],speeddata0,DefaultBlend,tool0;
  MoveAbsJ [[151.76,-36.67,-163.09,-53.47,-68.41,14.89],[9E9,9E9,9E9,9E9,9E9,9E9]],speeddata0,DefaultBlend,tool0;
  MoveAbsJ [[151.43,-36.51,-163.47,-54.46,-68.16,15.36],[9E9,9E9,9E9,9E9,9E9,9E9]],speeddata0,DefaultBlend,tool0;
  MoveAbsJ [[151.10,-36.34,-163.84,-55.45,-67.91,15.83],[9E9,9E9,9E9,9E9,9E9,9E9]],speeddata0,DefaultBlend,tool0;
  MoveAbsJ [[150.77,-36.18,-164.22,-56.44,-67.66,16.30],[9E9,9E9,9E9,9E9,9E9,9E9]],speeddata0,DefaultBlend,tool0;
  MoveAbsJ [[150.44,-36.02,-164.60,-57.43,-67.41,16.77],[9E9,9E9,9E9,9E9,9E9,9E9]],speeddata0,DefaultBlend,tool0;
  MoveAbsJ [[150.12,-35.85,-164.98,-58.42,-67.16,17.24],[9E9,9E9,9E9,9E9,9E9,9E9]],speeddata0,DefaultBlend,tool0;
  MoveAbsJ [[149.79,-35.69,-165.35,-59.41,-66.91,17.71],[9E9,9E9,9E9,9E9,9E9,9E9]],speeddata0,DefaultBlend,tool0;
  MoveAbsJ [[149.46,-35.53,-165.73,-60.40,-66.67,18.18],[9E9,9E9,9E9,9E9,9E9,9E9]],speeddata0,DefaultBlend,tool0;
  MoveAbsJ [[149.13,-35.37,-166.11,-61.39,-66.42,18.65],[9E9,9E9,9E9,9E9,9E9,9E9]],speeddata0,DefaultBlend,tool0;
  MoveAbsJ [[148.80,-35.20,-166.49,-62.38,-66.17,19.12],[9E9,9E9,9E9,9E9,9E9,9E9]],speeddata0,DefaultBlend,tool0;
  MoveAbsJ [[148.47,-35.04,-166.86,-63.37,-65.92,19.59],[9E9,9E9,9E9,9E9,9E9,9E9]],speeddata0,DefaultBlend,tool0;
  MoveAbsJ [[148.14,-34.88,-167.24,-64.36,-65.67,20.06],[9E9,9E9,9E9,9E9,9E9,9E9]],speeddata0,DefaultBlend,tool0;
  MoveAbsJ [[147.82,-34.72,-167.62,-65.35,-65.42,20.53],[9E9,9E9,9E9,9E9,9E9,9E9]],speeddata0,DefaultBlend,tool0;
  MoveAbsJ [[147.49,-34.55,-168.00,-66.34,-65.17,21.00],[9E9,9E9,9E9,9E9,9E9,9E9]],speeddata0,DefaultBlend,tool0;
  MoveAbsJ [[147.16,-34.39,-168.37,-67.33,-64.92,21.47],[9E9,9E9,9E9,9E9,9E9,9E9]],speeddata0,DefaultBlend,tool0;
  MoveAbsJ [[146.83,-34.23,-168.75,-68.32,-64.67,21.94],[9E9,9E9,9E9,9E9,9E9,9E9]],speeddata0,DefaultBlend,tool0;
  MoveAbsJ [[146.50,-34.06,-169.13,-69.32,-64.43,22.41],[9E9,9E9,9E9,9E9,9E9,9E9]],speeddata0,DefaultBlend,tool0;
  MoveAbsJ [[146.17,-33.90,-169.51,-70.31,-64.18,22.88],[9E9,9E9,9E9,9E9,9E9,9E9]],speeddata0,DefaultBlend,tool0;
  MoveAbsJ [[145.84,-33.74,-169.89,-71.30,-63.93,23.35],[9E9,9E9,9E9,9E9,9E9,9E9]],speeddata0,DefaultBlend,tool0;
  MoveAbsJ [[145.51,-33.58,-170.26,-72.29,-63.68,23.82],[9E9,9E9,9E9,9E9,9E9,9E9]],speeddata0,DefaultBlend,tool0;
  MoveAbsJ [[145.19,-33.41,-170.64,-73.28,-63.43,24.29],[9E9,9E9,9E9,9E9,9E9,9E9]],speeddata0,DefaultBlend,tool0;
  MoveAbsJ [[144.86,-33.25,-171.02,-74.27,-63.18,24.76],[9E9,9E9,9E9,9E9,9E9,9E9]],speeddata0,DefaultBlend,tool0;
  MoveAbsJ [[144.53,-33.09,-171.40,-75.26,-62.93,25.23],[9E9,9E9,9E9,9E9,9E9,9E9]],speeddata0,DefaultBlend,tool0;
  MoveAbsJ [[144.20,-32.93,-171.77,-76.25,-62.68,25.70],[9E9,9E9,9E9,9E9,9E9,9E9]],speeddata0,DefaultBlend,tool0;
  MoveAbsJ [[143.87,-32.76,-172.15,-77.24,-62.43,26.17],[9E9,9E9,9E9,9E9,9E9,9E9]],speeddata0,DefaultBlend,tool0;
  MoveAbsJ [[143.54,-32.60,-172.53,-78.23,-62.19,26.64],[9E9,9E9,9E9,9E9,9E9,9E9]],speeddata0,DefaultBlend,tool0;
  MoveAbsJ [[143.21,-32.44,-172.91,-79.22,-61.94,27.11],[9E9,9E9,9E9,9E9,9E9,9E9]],speeddata0,DefaultBlend,tool0;
  MoveAbsJ [[142.88,-32.27,-173.28,-80.21,-61.69,27.58],[9E9,9E9,9E9,9E9,9E9,9E9]],speeddata0,DefaultBlend,tool0;
  MoveAbsJ [[142.56,-32.11,-173.66,-81.20,-61.44,28.05],[9E9,9E9,9E9,9E9,9E9,9E9]],speeddata0,DefaultBlend,tool0;
  MoveAbsJ [[142.23,-31.95,-174.04,-82.19,-61.19,28.52],[9E9,9E9,9E9,9E9,9E9,9E9]],speeddata0,DefaultBlend,tool0;
  MoveAbsJ [[141.90,-31.79,-174.42,-83.18,-60.94,28.99],[9E9,9E9,9E9,9E9,9E9,9E9]],speeddata0,DefaultBlend,tool0;
  MoveAbsJ [[141.57,-31.62,-174.79,-84.17,-60.69,29.46],[9E9,9E9,9E9,9E9,9E9,9E9]],speeddata0,DefaultBlend,tool0;
  MoveAbsJ [[141.24,-31.46,-175.17,-85.16,-60.44,29.93],[9E9,9E9,9E9,9E9,9E9,9E9]],speeddata0,DefaultBlend,tool0;
  MoveAbsJ [[140.91,-31.30,-175.55,-86.15,-60.19,30.40],[9E9,9E9,9E9,9E9,9E9,9E9]],speeddata0,DefaultBlend,tool0;
  MoveAbsJ [[140.58,-31.14,-175.93,-87.14,-59.95,30.87],[9E9,9E9,9E9,9E9,9E9,9E9]],speeddata0,DefaultBlend,tool0;
  MoveAbsJ [[140.26,-30.97,-176.30,-88.13,-59.70,31.34],[9E9,9E9,9E9,9E9,9E9,9E9]],speeddata0,DefaultBlend,tool0;
  MoveAbsJ [[139.93,-30.81,-176.68,-89.12,-59.45,31.81],[9E9,9E9,9E9,9E9,9E9,9E9]],speeddata0,DefaultBlend,tool0;
  MoveAbsJ [[139.60,-30.65,-177.06,-90.11,-59.20,32.28],[9E9,9E9,9E9,9E9,9E9,9E9]],speeddata0,DefaultBlend,tool0;
  MoveAbsJ [[139.27,-30.48,-177.44,-91.10,-58.95,32.75],[9E9,9E9,9E9,9E9,9E9,9E9]],speeddata0,DefaultBlend,tool0;
  MoveAbsJ [[138.94,-30.32,-177.82,-92.09,-58.70,33.22],[9E9,9E9,9E9,9E9,9E9,9E9]],speeddata0,DefaultBlend,tool0;
  MoveAbsJ [[138.61,-30.16,-178.19,-93.08,-58.45,33.69],[9E9,9E9,9E9,9E9,9E9,9E9]],speeddata0,DefaultBlend,tool0;
  MoveAbsJ [[138.28,-30.00,-178.57,-94.07,-58.20,34.16],[9E9,9E9,9E9,9E9,9E9,9E9]],speeddata0,DefaultBlend,tool0;
  MoveAbsJ [[137.95,-29.83,-178.95,-95.06,-57.95,34.63],[9E9,9E9,9E9,9E9,9E9,9E9]],speeddata0,DefaultBlend,tool0;
  MoveAbsJ [[137.63,-29.67,-179.33,-96.05,-57.71,35.10],[9E9,9E9,9E9,9E9,9E9,9E9]],speeddata0,DefaultBlend,tool0;
  MoveAbsJ [[137.30,-29.51,-179.70,-97.04,-57.46,35.57],[9E9,9E9,9E9,9E9,9E9,9E9]],speeddata0,DefaultBlend,tool0;
  MoveAbsJ [[136.97,-29.35,-180.08,-98.03,-57.21,36.04],[9E9,9E9,9E9,9E9,9E9,9E9]],speeddata0,DefaultBlend,tool0;
  MoveAbsJ [[136.64,-29.18,-180.46,-99.02,-56.96,36.51],[9E9,9E9,9E9,9E9,9E9,9E9]],speeddata0,DefaultBlend,tool0;
  MoveAbsJ [[136.31,-29.02,-180.84,-100.01,-56.71,36.98],[9E9,9E9,9E9,9E9,9E9,9E9]],speeddata0,DefaultBlend,tool0;
  MoveAbsJ [[135.98,-28.86,-181.21,-101.00,-56.46,37.45],[9E9,9E9,9E9,9E9,9E9,9E9]],speeddata0,DefaultBlend,tool0;
  MoveAbsJ [[135.65,-28.69,-181.59,-101.99,-56.21,37.92],[9E9,9E9,9E9,9E9,9E9,9E9]],speeddata0,DefaultBlend,tool0;
  MoveAbsJ [[135.32,-28.53,-181.97,-102.98,-55.96,38.39],[9E9,9E9,9E9,9E9,9E9,9E9]],speeddata0,DefaultBlend,tool0;
  MoveAbsJ [[135.00,-28.37,-182.35,-103.97,-55.71,38.86],[9E9,9E9,9E9,9E9,9E9,9E9]],speeddata0,DefaultBlend,tool0;
  MoveAbsJ [[134.67,-28.21,-182.72,-104.96,-55.47,39.33],[9E9,9E9,9E9,9E9,9E9,9E9]],speeddata0,DefaultBlend,tool0;
  MoveAbsJ [[134.34,-28.04,-183.10,-105.95,-55.22,39.80],[9E9,9E9,9E9,9E9,9E9,9E9]],speeddata0,DefaultBlend,tool0;
  MoveAbsJ [[134.01,-27.88,-183.48,-106.94,-54.97,40.27],[9E9,9E9,9E9,9E9,9E9,9E9]],speeddata0,DefaultBlend,tool0;
  MoveAbsJ [[133.68,-27.72,-183.86,-107.93,-54.72,40.74],[9E9,9E9,9E9,9E9,9E9,9E9]],speeddata0,DefaultBlend,tool0;
  MoveAbsJ [[133.35,-27.56,-184.24,-108.92,-54.47,41.21],[9E9,9E9,9E9,9E9,9E9,9E9]],speeddata0,DefaultBlend,tool0;
  MoveAbsJ [[133.02,-27.39,-184.61,-109.91,-54.22,41.68],[9E9,9E9,9E9,9E9,9E9,9E9]],speeddata0,DefaultBlend,tool0;
  MoveAbsJ [[132.70,-27.23,-184.99,-110.90,-53.97,42.15],[9E9,9E9,9E9,9E9,9E9,9E9]],speeddata0,DefaultBlend,tool0;
  MoveAbsJ [[132.37,-27.07,-185.37,-111.89,-53.72,42.62],[9E9,9E9,9E9,9E9,9E9,9E9]],speeddata0,DefaultBlend,tool0;
  MoveAbsJ [[132.04,-26.90,-185.75,-112.88,-53.47,43.09],[9E9,9E9,9E9,9E9,9E9,9E9]],speeddata0,DefaultBlend,tool0;
  MoveAbsJ [[131.71,-26.74,-186.12,-113.87,-53.23,43.56],[9E9,9E9,9E9,9E9,9E9,9E9]],speeddata0,DefaultBlend,tool0;
  MoveAbsJ [[131.38,-26.58,-186.50,-114.87,-52.98,44.03],[9E9,9E9,9E9,9E9,9E9,9E9]],speeddata0,DefaultBlend,tool0;
  MoveAbsJ [[131.05,-26.42,-186.88,-115.86,-52.73,44.50],[9E9,9E9,9E9,9E9,9E9,9E9]],speeddata0,DefaultBlend,tool0;
  MoveAbsJ [[130.72,-26.25,-187.26,-116.85,-52.48,44.97],[9E9,9E9,9E9,9E9,9E9,9E9]],speeddata0,DefaultBlend,tool0;
  MoveAbsJ [[130.39,-26.09,-187.63,-117.84,-52.23,45.44],[9E9,9E9,9E9,9E9,9E9,9E9]],speeddata0,DefaultBlend,tool0;
  MoveAbsJ [[130.07,-25.93,-188.01,-118.83,-51.98,45.91],[9E9,9E9,9E9,9E9,9E9,9E9]],speeddata0,DefaultBlend,tool0;
  MoveAbsJ [[129.74,-25.77,-188.39,-119.82,-51.73,46.38],[9E9,9E9,9E9,9E9,9E9,9E9]],speeddata0,DefaultBlend,tool0;
  MoveAbsJ [[129.41,-25.60,-188.77,-120.81,-51.48,46.85],[9E9,9E9,9E9,9E9,9E9,9E9]],speeddata0,DefaultBlend,tool0;
  MoveAbsJ [[129.08,-25.44,-189.14,-121.80,-51.23,47.32],[9E9,9E9,9E9,9E9,9E9,9E9]],speeddata0,DefaultBlend,tool0;
  MoveAbsJ [[128.75,-25.28,-189.52,-122.79,-50.99,47.79],[9E9,9E9,9E9,9E9,9E9,9E9]],speeddata0,DefaultBlend,tool0;
  MoveAbsJ [[128.42,-25.11,-189.90,-123.78,-50.74,48.26],[9E9,9E9,9E9,9E9,9E9,9E9]],speeddata0,DefaultBlend,tool0;
  MoveAbsJ [[128.09,-24.95,-190.28,-124.77,-50.49,48.73],[9E9,9E9,9E9,9E9,9E9,9E9]],speeddata0,DefaultBlend,tool0;
  MoveAbsJ [[127.77,-24.79,-190.66,-125.76,-50.24,49.20],[9E9,9E9,9E9,9E9,9E9,9E9]],speeddata0,DefaultBlend,tool0;
  MoveAbsJ [[127.44,-24.63,-191.03,-126.75,-49.99,49.67],[9E9,9E9,9E9,9E9,9E9,9E9]],speeddata0,DefaultBlend,tool0;
  MoveAbsJ [[127.11,-24.46,-191.41,-127.74,-49.74,50.14],[9E9,9E9,9E9,9E9,9E9,9E9]],speeddata0,FinePoint,tool0;
  TPWrite "Action 36 LoadWorkpiece.";
  TPWrite "Press Play to Continue";
  Stop;
  TPWrite "Action 37 CloseGripper.";
  TPWrite "Press Play to Continue";
  Stop;
  TPWrite "Action 38 FreeMovement.";
  MoveAbsJ [[127.11,-24.46,-191.41,-127.74,-49.74,50.14],[9E9,9E9,9E9,9E9,9E9,9E9]],speeddata0,DefaultBlend,tool0;
  MoveAbsJ [[126.60,-24.25,-190.42,-127.91,-49.27,49.88],[9E9,9E9,9E9,9E9,9E9,9E9]],speeddata0,DefaultBlend,tool0;
  MoveAbsJ [[126.08,-24.04,-189.43,-128.07,-48.81,49.62],[9E9,9E9,9E9,9E9,9E9,9E9]],speeddata0,DefaultBlend,tool0;
  MoveAbsJ [[125.57,-23.83,-188.44,-128.24,-48.34,49.36],[9E9,9E9,9E9,9E9,9E9,9E9]],speeddata0,DefaultBlend,tool0;
  MoveAbsJ [[125.06,-23.62,-187.45,-128.41,-47.87,49.10],[9E9,9E9,9E9,9E9,9E9,9E9]],speeddata0,DefaultBlend,tool0;
  MoveAbsJ [[124.55,-23.42,-186.45,-128.58,-47.41,48.84],[9E9,9E9,9E9,9E9,9E9,9E9]],speeddata0,DefaultBlend,tool0;
  MoveAbsJ [[124.04,-23.21,-185.46,-128.74,-46.94,48.58],[9E9,9E9,9E9,9E9,9E9,9E9]],speeddata0,DefaultBlend,tool0;
  MoveAbsJ [[123.52,-23.00,-184.47,-128.91,-46.48,48.32],[9E9,9E9,9E9,9E9,9E9,9E9]],speeddata0,DefaultBlend,tool0;
  MoveAbsJ [[123.01,-22.79,-183.48,-129.08,-46.01,48.06],[9E9,9E9,9E9,9E9,9E9,9E9]],speeddata0,DefaultBlend,tool0;
  MoveAbsJ [[122.50,-22.58,-182.49,-129.25,-45.54,47.80],[9E9,9E9,9E9,9E9,9E9,9E9]],speeddata0,DefaultBlend,tool0;
  MoveAbsJ [[121.99,-22.37,-181.50,-129.41,-45.08,47.54],[9E9,9E9,9E9,9E9,9E9,9E9]],speeddata0,DefaultBlend,tool0;
  MoveAbsJ [[121.48,-22.16,-180.51,-129.58,-44.61,47.28],[9E9,9E9,9E9,9E9,9E9,9E9]],speeddata0,DefaultBlend,tool0;
  MoveAbsJ [[120.96,-21.95,-179.51,-129.75,-44.14,47.02],[9E9,9E9,9E9,9E9,9E9,9E9]],speeddata0,DefaultBlend,tool0;
  MoveAbsJ [[120.45,-21.74,-178.52,-129.92,-43.68,46.76],[9E9,9E9,9E9,9E9,9E9,9E9]],speeddata0,DefaultBlend,tool0;
  MoveAbsJ [[119.94,-21.53,-177.53,-130.09,-43.21,46.50],[9E9,9E9,9E9,9E9,9E9,9E9]],speeddata0,DefaultBlend,tool0;
  MoveAbsJ [[119.43,-21.32,-176.54,-130.25,-42.74,46.24],[9E9,9E9,9E9,9E9,9E9,9E9]],speeddata0,DefaultBlend,tool0;
  MoveAbsJ [[118.92,-21.11,-175.55,-130.42,-42.28,45.98],[9E9,9E9,9E9,9E9,9E9,9E9]],speeddata0,DefaultBlend,tool0;
  MoveAbsJ [[118.40,-20.90,-174.56,-130.59,-41.81,45.72],[9E9,9E9,9E9,9E9,9E9,9E9]],speeddata0,DefaultBlend,tool0;
  MoveAbsJ [[117.89,-20.69,-173.57,-130.76,-41.34,45.46],[9E9,9E9,9E9,9E9,9E9,9E9]],speeddata0,DefaultBlend,tool0;
  MoveAbsJ [[117.38,-20.48,-172.58,-130.92,-40.88,45.20],[9E9,9E9,9E9,9E9,9E9,9E9]],speeddata0,DefaultBlend,tool0;
  MoveAbsJ [[116.87,-20.27,-171.58,-131.09,-40.41,44.94],[9E9,9E9,9E9,9E9,9E9,9E9]],speeddata0,DefaultBlend,tool0;
  MoveAbsJ [[116.36,-20.06,-170.59,-131.26,-39.94,44.68],[9E9,9E9,9E9,9E9,9E9,9E9]],speeddata0,DefaultBlend,tool0;
  MoveAbsJ [[115.84,-19.85,-169.60,-131.43,-39.48,44.42],[9E9,9E9,9E9,9E9,9E9,9E9]],speeddata0,DefaultBlend,tool0;
  MoveAbsJ [[115.33,-19.64,-168.61,-131.59,-39.01,44.16],[9E9,9E9,9E9,9E9,9E9,9E9]],speeddata0,DefaultBlend,tool0;
  MoveAbsJ [[114.82,-19.43,-167.62,-131.76,-38.54,43.90],[9E9,9E9,9E9,9E9,9E9,9E9]],speeddata0,DefaultBlend,tool0;
  MoveAbsJ [[114.31,-19.22,-166.63,-131.93,-38.08,43.64],[9E9,9E9,9E9,9E9,9E9,9E9]],speeddata0,DefaultBlend,tool0;
  MoveAbsJ [[113.79,-19.01,-165.64,-132.10,-37.61,43.38],[9E9,9E9,9E9,9E9,9E9,9E9]],speeddata0,DefaultBlend,tool0;
  MoveAbsJ [[113.28,-18.80,-164.64,-132.26,-37.14,43.12],[9E9,9E9,9E9,9E9,9E9,9E9]],speeddata0,DefaultBlend,tool0;
  MoveAbsJ [[112.77,-18.59,-163.65,-132.43,-36.68,42.86],[9E9,9E9,9E9,9E9,9E9,9E9]],speeddata0,DefaultBlend,tool0;
  MoveAbsJ [[112.26,-18.38,-162.66,-132.60,-36.21,42.60],[9E9,9E9,9E9,9E9,9E9,9E9]],speeddata0,DefaultBlend,tool0;
  MoveAbsJ [[111.75,-18.17,-161.67,-132.77,-35.74,42.34],[9E9,9E9,9E9,9E9,9E9,9E9]],speeddata0,DefaultBlend,tool0;
  MoveAbsJ [[111.23,-17.96,-160.68,-132.94,-35.28,42.08],[9E9,9E9,9E9,9E9,9E9,9E9]],speeddata0,DefaultBlend,tool0;
  MoveAbsJ [[110.72,-17.75,-159.69,-133.10,-34.81,41.82],[9E9,9E9,9E9,9E9,9E9,9E9]],speeddata0,DefaultBlend,tool0;
  MoveAbsJ [[110.21,-17.54,-158.70,-133.27,-34.34,41.55],[9E9,9E9,9E9,9E9,9E9,9E9]],speeddata0,DefaultBlend,tool0;
  MoveAbsJ [[109.70,-17.33,-157.70,-133.44,-33.88,41.29],[9E9,9E9,9E9,9E9,9E9,9E9]],speeddata0,DefaultBlend,tool0;
  MoveAbsJ [[109.19,-17.12,-156.71,-133.61,-33.41,41.03],[9E9,9E9,9E9,9E9,9E9,9E9]],speeddata0,DefaultBlend,tool0;
  MoveAbsJ [[108.67,-16.92,-155.72,-133.77,-32.94,40.77],[9E9,9E9,9E9,9E9,9E9,9E9]],speeddata0,DefaultBlend,tool0;
  MoveAbsJ [[108.16,-16.71,-154.73,-133.94,-32.48,40.51],[9E9,9E9,9E9,9E9,9E9,9E9]],speeddata0,DefaultBlend,tool0;
  MoveAbsJ [[107.65,-16.50,-153.74,-134.11,-32.01,40.25],[9E9,9E9,9E9,9E9,9E9,9E9]],speeddata0,DefaultBlend,tool0;
  MoveAbsJ [[107.14,-16.29,-152.75,-134.28,-31.54,39.99],[9E9,9E9,9E9,9E9,9E9,9E9]],speeddata0,DefaultBlend,tool0;
  MoveAbsJ [[106.63,-16.08,-151.76,-134.44,-31.08,39.73],[9E9,9E9,9E9,9E9,9E9,9E9]],speeddata0,DefaultBlend,tool0;
  MoveAbsJ [[106.11,-15.87,-150.77,-134.61,-30.61,39.47],[9E9,9E9,9E9,9E9,9E9,9E9]],speeddata0,DefaultBlend,tool0;
  MoveAbsJ [[105.60,-15.66,-149.77,-134.78,-30.14,39.21],[9E9,9E9,9E9,9E9,9E9,9E9]],speeddata0,DefaultBlend,tool0;
  MoveAbsJ [[105.09,-15.45,-148.78,-134.95,-29.68,38.95],[9E9,9E9,9E9,9E9,9E9,9E9]],speeddata0,DefaultBlend,tool0;
  MoveAbsJ [[104.58,-15.24,-147.79,-135.11,-29.21,38.69],[9E9,9E9,9E9,9E9,9E9,9E9]],speeddata0,DefaultBlend,tool0;
  MoveAbsJ [[104.07,-15.03,-146.80,-135.28,-28.74,38.43],[9E9,9E9,9E9,9E9,9E9,9E9]],speeddata0,DefaultBlend,tool0;
  MoveAbsJ [[103.55,-14.82,-145.81,-135.45,-28.28,38.17],[9E9,9E9,9E9,9E9,9E9,9E9]],speeddata0,DefaultBlend,tool0;
  MoveAbsJ [[103.04,-14.61,-144.82,-135.62,-27.81,37.91],[9E9,9E9,9E9,9E9,9E9,9E9]],speeddata0,DefaultBlend,tool0;
  MoveAbsJ [[102.53,-14.40,-143.83,-135.79,-27.34,37.65],[9E9,9E9,9E9,9E9,9E9,9E9]],speeddata0,DefaultBlend,tool0;
